// TwinCAT 3 PLC project DataProcessing
// ProgramVersion: 3.1.4023.0
// libraries:
//   Tc2_Standard, * (Beckhoff Automation GmbH)
//   Tc2_System, * (Beckhoff Automation GmbH)
//   Tc2_Utilities, * (Beckhoff Automation GmbH)
//   Tc3_EventLogger, * (Beckhoff Automation GmbH)
//   Tc3_Module, * (Beckhoff Automation GmbH)
// project tree:
//   DUTs/ FB_GetFaultWordsFromProtxConverter.TcPOU, FB_PrepareOutputVectorsToProTxConverter.TcPOU, FB_PrepareInputVectorsFromProTxCovnerter.TcPOU, FB_GetStatusWordsFromProTxConverter.TcPOU
//   Enumerations/ E_DriveProfile.TcDUT
//   EventLogger/FunctionBlocks/Common/ P_EventLogger.TcPOU, P_Timer.TcPOU
//   EventLogger/FunctionBlocks/ FB_EventMessage.TcPOU, FB_EventAlarm.TcPOU
//   GVLs/ ConfigurationParameters.TcGVL, RxAndTxData.TcGVL, StatusAndCommandWordsStructures.TcGVL, UtilityVariables.TcGVL
//   GVLs/ST_OutputVectorsToProTx/ ST_OutputVectorReal.TcDUT, ST_LcCommandWord_ProfiDrive.TcDUT, ST_McCommandWord_1_ProfiDrive.TcDUT, ST_McCommandWord_2_ProfiDrive.TcDUT
//   GVLs/ST_InputVectorsFromProTx/ST_FaultWords/ ST_LcFaultWord1.TcDUT, ST_LcFaultWord2.TcDUT, ST_LcFaultWord3.TcDUT, ST_LcFaultWord4.TcDUT, ST_McFaultWord1.TcDUT, ST_McFaultWord2.TcDUT, ST_McFaultWord3.TcDUT, ST_McFaultWord4.TcDUT
//   GVLs/ST_InputVectorsFromProTx/ ST_LcStatusWord_2_ProfiDrive.TcDUT, ST_McStatusWord_2_ProfiDrive.TcDUT, ST_LcStatusWord_1_ProfiDrive.TcDUT, ST_McStatusWord_1_ProfiDrive.TcDUT, ST_OutputVectorReal1.TcDUT
//   / PlcTask.TcTTO
//   POUs/ MAIN.TcPOU
// real-time tasks:
//   TASK PlcTask: cycle T#1ms, priority 20, ADS port 350

CONFIGURATION DataProcessing
    RESOURCE PLC ON TwinCAT3
        TASK PlcTask(INTERVAL := T#1ms, PRIORITY := 20);
        PROGRAM MAIN WITH PlcTask : MAIN;
    END_RESOURCE
END_CONFIGURATION

// ---- Enumerations/E_DriveProfile.TcDUT
{attribute 'qualified_only'}
{attribute 'strict'}
TYPE E_DriveProfile :
(
	CiA402 		:= 1,
	CAN 		:= 2,
	ProfiDrive  := 3
	
) := ProfiDrive;
END_TYPE

// ---- GVLs/ST_OutputVectorsToProTx/ST_OutputVectorReal.TcDUT
TYPE ST_OutputVectorReal :
STRUCT
	OutputPDO_1 			: REAL; // LC Iq_ref and  MC torque or current
	OutputPDO_2 			: REAL; // MC speed or voltge
	OutputPDO_3				: REAL; // Mc act. torque or power
	OutputPDO_4				: REAL; // MC Ext Torque Limmit_motor or Charge current limmit
	OutputPDO_5				: REAL; // MC Ext Torque Limmit_gen or Discharge current limmit
	OutputPDO_6				: REAL; // MC Speed regulation bias and Cable resistor in Ohm
	OutputPDO_7				: REAL; // MC Speed limmit and Max output votltage switch off value in V
	OutputPDO_8				: REAL; // MC Jrequest and and Min output votltage switch off value in V
	OutputPDO_9				: REAL; // MC Max output current switch off value in A and ETPS value for number of cylinders
	OutputPDO_10			: REAL;	// MC Min output current switch off value in A and scaled ETPS torque M1
END_STRUCT
END_TYPE

// ---- GVLs/ST_OutputVectorsToProTx/ST_LcCommandWord_ProfiDrive.TcDUT
TYPE ST_LcCommandWord_ProfiDrive :
STRUCT
	Bit00_OnOff 						: BOOL;
	Bit01_DriveRelease					: BOOL;
	Bit02_uu 							: BOOL;
	Bit03_PulseRelease 					: BOOL;
	Bit04_uu							: BOOL;
	Bit05_uu							: BOOL;
	Bit06_uu							: BOOL;
	Bit07_Quit							: BOOL;
	Bit08_uu							: BOOL;
	Bit09_uu							: BOOL;
	Bit10_ControlByPLC					: BOOL;
	Bit11_ParSetChangeOverBit00			: BOOL;
	Bit12_ParSetChangeOverBit01			: BOOL;
	Bit13_ParSetChangeOverBit02			: BOOL;
	Bit14_ParSetChangeOverBit03			: BOOL;
	Bit15_MainAliveToggle				: BOOL;

END_STRUCT
END_TYPE

// ---- GVLs/ST_OutputVectorsToProTx/ST_McCommandWord_1_ProfiDrive.TcDUT
TYPE ST_McCommandWord_1_ProfiDrive :
STRUCT
	Bit00_OnOff 					: BOOL;
	Bit01_DriveRelease				: BOOL;
	Bit02_FastStop 					: BOOL; // FALCE - forces QuickStop
	Bit03_PulceRelease 				: BOOL;
	Bit04_EnableRump				: BOOL; // TRUE - Select ramp output as reference; FALCE - select other reference source - may be zero 
	Bit05_UnlockRump				: BOOL; // TRUE - Ramp output shall follow ramp input; FALCE - Ramp output shall be locked to current output value
	Bit06_Forward					: BOOL;
	Bit07_Quit						: BOOL;
	Bit08_Inching1					: BOOL;
	Bit09_Inching2					: BOOL;
	Bit10_ControlByPlc				: BOOL;
	Bit11_ParSetChangeOverBit00		: BOOL;
	Bit12_ParSetChangeOverBit01		: BOOL;
	Bit13_ParSetChangeOverBit02		: BOOL;
	Bit14_ParSetChangeOverBit03		: BOOL;
	Bit15_MainAliveToggle			: BOOL;	
END_STRUCT
END_TYPE

// ---- GVLs/ST_OutputVectorsToProTx/ST_McCommandWord_2_ProfiDrive.TcDUT
TYPE ST_McCommandWord_2_ProfiDrive :
STRUCT
	Bit00_IntegratorSpeedCtrlDisable	: BOOL;
	Bit01_TorqueControlModeActive		: BOOL;
	Bit02_GainSpeedcontrolChangeover 	: BOOL;
	Bit03_Drooping 						: BOOL;
	Bit04_TorqueControlEnable			: BOOL;
	Bit05_TorqueReferenceEnable			: BOOL;
	Bit06_EtpsEnable					: BOOL;
	Bit07_EtpsInputSourceSelect			: BOOL;
	Bit08_InertiaCompensationenable		: BOOL;
	Bit09_ExternalMotorFanOff			: BOOL;
	Bit10_uu							: BOOL;
	Bit11_uu							: BOOL;
	Bit12_Reverce						: BOOL;
	Bit13_BrakeControl					: BOOL;
	Bit14_BrakeTestMode					: BOOL;
	Bit15_InternalAliveToggle			: BOOL;	
END_STRUCT
END_TYPE

// ---- GVLs/ST_InputVectorsFromProTx/ST_FaultWords/ST_LcFaultWord1.TcDUT
TYPE ST_LcFaultWord1 :
STRUCT
	Bit00_FaultInputAryEcat 	: BOOL;
	Bit01_FPGA					: BOOL;
	Bit02_Watchdog 				: BOOL;
	Bit03_UdcMax 				: BOOL;
	Bit04_uu					: BOOL;
	Bit05_uu					: BOOL;
	Bit06_uu					: BOOL;
	Bit07_uu					: BOOL;
	Bit08_UceFault				: BOOL;
	Bit09_uu					: BOOL;
	Bit10_uu					: BOOL;
	Bit11_uu					: BOOL;
	Bit12_uu					: BOOL;
	Bit13_uu					: BOOL;
	Bit14_uu					: BOOL;
	Bit15_uu					: BOOL;	
END_STRUCT
END_TYPE

// ---- GVLs/ST_InputVectorsFromProTx/ST_FaultWords/ST_LcFaultWord2.TcDUT
TYPE ST_LcFaultWord2 :
STRUCT
	Bit00_PibSupply 				: BOOL;
	Bit01_MeasurementConnectorLoop	: BOOL;
	Bit02_FaultLoop 				: BOOL;
	Bit03_AmplifierConnector 		: BOOL;
	Bit04_TermSupply 				: BOOL;
	Bit05_Overcurrent 				: BOOL;
	Bit06_ShortCircuit 				: BOOL;
	Bit07_DcConnection				: BOOL;
	Bit08_ThHSMax					: BOOL;
	Bit09_ShortCircuit24V			: BOOL;
	Bit10_FieldBus					: BOOL;
	Bit11_FLinkRxMc					: BOOL;
	Bit12_EarthFault				: BOOL;
	Bit13_UdcMin					: BOOL;
	Bit14_uu						: BOOL;
	Bit15_ExtFault					: BOOL;	
END_STRUCT
END_TYPE

// ---- GVLs/ST_InputVectorsFromProTx/ST_FaultWords/ST_LcFaultWord3.TcDUT
TYPE ST_LcFaultWord3 :
STRUCT
	Bit00_ULineVoltage 				: BOOL;
	Bit01_ULineMeasurement			: BOOL;
	Bit02_AcFuse	 				: BOOL;
	Bit03_FbLineContactor	 		: BOOL;
	Bit04_Charging	 				: BOOL;
	Bit05_LineFilter 				: BOOL;
	Bit06_uu		 				: BOOL;
	Bit07_uu						: BOOL;
	Bit08_uu						: BOOL;
	Bit09_uu						: BOOL;
	Bit10_uu						: BOOL;
	Bit11_uu						: BOOL;
	Bit12_uu						: BOOL;
	Bit13_uu						: BOOL;
	Bit14_uu						: BOOL;
	Bit15_uu						: BOOL;	
END_STRUCT
END_TYPE

// ---- GVLs/ST_InputVectorsFromProTx/ST_FaultWords/ST_LcFaultWord4.TcDUT
TYPE ST_LcFaultWord4 :
STRUCT
	Bit00_NTC 						: BOOL;
	Bit01_ThHsMin					: BOOL;
	Bit02_CoolingSystem 			: BOOL;
	Bit03_ControllerCabinetFan 		: BOOL;
	Bit04_ConverterCubiceOvertemp 	: BOOL;
	Bit05_CubicleAuxSupply 			: BOOL;
	Bit06_uu 						: BOOL;
	Bit07_uu						: BOOL;
	Bit08_uu						: BOOL;
	Bit09_FeedInCubicleOvertemp		: BOOL;
	Bit10_TrafoOvertemp				: BOOL;
	Bit11_Isolation					: BOOL;
	Bit12_uu						: BOOL;
	Bit13_uu						: BOOL;
	Bit14_uu						: BOOL;
	Bit15_uu						: BOOL;	
END_STRUCT
END_TYPE

// ---- GVLs/ST_InputVectorsFromProTx/ST_FaultWords/ST_McFaultWord1.TcDUT
TYPE ST_McFaultWord1 :
STRUCT
	Bit00_FaultInputAryEcat 	: BOOL;
	Bit01_FPGA					: BOOL;
	Bit02_Watchdog 				: BOOL;
	Bit03_UdcMax 				: BOOL;
	Bit04_uu					: BOOL;
	Bit05_uu					: BOOL;
	Bit06_uu					: BOOL;
	Bit07_uu					: BOOL;
	Bit08_UceFault				: BOOL;
	Bit09_uu					: BOOL;
	Bit10_uu					: BOOL;
	Bit11_uu					: BOOL;
	Bit12_uu					: BOOL;
	Bit13_uu					: BOOL;
	Bit14_uu					: BOOL;
	Bit15_uu					: BOOL;	
END_STRUCT
END_TYPE

// ---- GVLs/ST_InputVectorsFromProTx/ST_FaultWords/ST_McFaultWord2.TcDUT
TYPE ST_McFaultWord2 :
STRUCT
	Bit00_PibSupply 				: BOOL;
	Bit01_MeasurementConnectorLoop	: BOOL;
	Bit02_FaultLoop 				: BOOL;
	Bit03_AmplifierConnector 		: BOOL;
	Bit04_TermSupply 				: BOOL;
	Bit05_Overcurrent 				: BOOL;
	Bit06_ShortCircuit 				: BOOL;
	Bit07_DcConnection				: BOOL;
	Bit08_ThHSMax					: BOOL;
	Bit09_ShortCircuit24V			: BOOL;
	Bit10_FieldBus					: BOOL;
	Bit11_FLinkRxMc					: BOOL;
	Bit12_EarthFault				: BOOL;
	Bit13_UdcMin					: BOOL;
	Bit14_uu						: BOOL;
	Bit15_ExtFault					: BOOL;	
END_STRUCT
END_TYPE

// ---- GVLs/ST_InputVectorsFromProTx/ST_FaultWords/ST_McFaultWord3.TcDUT
TYPE ST_McFaultWord3 :
STRUCT
	Bit00_EncoderFault 				: BOOL;
	Bit01_BlockFault				: BOOL;
	Bit02_OverspeedFault			: BOOL;
	Bit03_BrakeFault		 		: BOOL;
	Bit04_InterlockRotating			: BOOL;
	Bit05_DcOutputSwitches			: BOOL;
	Bit06_DcOutputOfRange			: BOOL;
	Bit07_DcSwitchOnSequence		: BOOL;
	Bit08_uu						: BOOL;
	Bit09_uu						: BOOL;
	Bit10_uu						: BOOL;
	Bit11_uu						: BOOL;
	Bit12_uu						: BOOL;
	Bit13_uu						: BOOL;
	Bit14_uu						: BOOL;
	Bit15_uu						: BOOL;	
END_STRUCT
END_TYPE

// ---- GVLs/ST_InputVectorsFromProTx/ST_FaultWords/ST_McFaultWord4.TcDUT
TYPE ST_McFaultWord4 :
STRUCT
	Bit00_NTC 						: BOOL;
	Bit01_ThHsMin					: BOOL;
	Bit02_uu			 			: BOOL;
	Bit03_ControllerCabinetFan 		: BOOL;
	Bit04_ConverterCubiceOvertemp 	: BOOL;
	Bit05_CubicleAuxSupply 			: BOOL;
	Bit06_MotorTemp					: BOOL;
	Bit07_uu						: BOOL;
	Bit08_FrequLock					: BOOL;
	Bit09_ConverterOverload			: BOOL;
	Bit10_uu						: BOOL;
	Bit11_uu						: BOOL;
	Bit12_uu						: BOOL;
	Bit13_uu						: BOOL;
	Bit14_uu						: BOOL;
	Bit15_uu						: BOOL;	
END_STRUCT
END_TYPE

// ---- GVLs/ST_InputVectorsFromProTx/ST_LcStatusWord_2_ProfiDrive.TcDUT
TYPE ST_LcStatusWord_2_ProfiDrive :
STRUCT
	Bit00_FaultB					: BOOL;
	Bit01_FaultC 					: BOOL;
	Bit02_FaultC 					: BOOL;
	Bit03_FaultDWarning 			: BOOL;
	Bit04_TrafoOvertempWarning		: BOOL;
	Bit05_TrafoInsolationWarning	: BOOL;
	Bit06_uu						: BOOL;
	Bit07_uu						: BOOL;
	Bit08_uu						: BOOL;
	Bit09_uu						: BOOL;
	Bit10_ThHSWarning				: BOOL;
	Bit11_ThHSMaxWarning			: BOOL;
	Bit12_ParSetBit00				: BOOL;
	Bit13_ParSetBit01				: BOOL;
	Bit14_ParSetBit02				: BOOL;
	Bit15_ParSetBit03				: BOOL;	
END_STRUCT
END_TYPE

// ---- GVLs/ST_InputVectorsFromProTx/ST_McStatusWord_2_ProfiDrive.TcDUT
TYPE ST_McStatusWord_2_ProfiDrive :
STRUCT
	Bit00_FaultB					: BOOL;
	Bit01_FaultC 					: BOOL;
	Bit02_FaultC 					: BOOL;
	Bit03_FaultDWarning 			: BOOL;
	Bit04_MRegActive				: BOOL;
	Bit05_torqueRegEnable			: BOOL;
	Bit06_ConverterI2tLinitWarning	: BOOL;
	Bit07_ConverterI2tLinitActive	: BOOL;
	Bit08_MotorI2tLinitWarning		: BOOL;
	Bit09_MotorI2tLinitActive		: BOOL;
	Bit10_ThHSWarning				: BOOL;
	Bit11_ThHSMaxWarning			: BOOL;
	Bit12_windingTempWarning		: BOOL;
	Bit13_BearingTempWarning		: BOOL;
	Bit14_Forward					: BOOL;
	Bit15_Reverse					: BOOL;	
END_STRUCT
END_TYPE

// ---- GVLs/ST_InputVectorsFromProTx/ST_LcStatusWord_1_ProfiDrive.TcDUT
TYPE ST_LcStatusWord_1_ProfiDrive :
STRUCT
	Bit00_StateReady			: BOOL;
	Bit01_StateOn 				: BOOL;
	Bit02_CtrlRun 				: BOOL;
	Bit03_CollFault 			: BOOL;
	Bit04_DriveReleaseActive	: BOOL;
	Bit05_StatePowerOk			: BOOL;
	Bit06_StateDisable			: BOOL;
	Bit07_Warning				: BOOL;
	Bit08_PhaseLoss				: BOOL;
	Bit09_BusSelected			: BOOL;
	Bit10_uu					: BOOL;
	Bit11_uu					: BOOL;
	Bit12_ReleaseMc				: BOOL;
	Bit13_StateTestModeOn		: BOOL;
	Bit14_InternalAliveToggle	: BOOL;
	Bit15_MainAliveToggle		: BOOL;	
END_STRUCT
END_TYPE

// ---- GVLs/ST_InputVectorsFromProTx/ST_McStatusWord_1_ProfiDrive.TcDUT
TYPE ST_McStatusWord_1_ProfiDrive :
STRUCT
	Bit00_StateReady			: BOOL;
	Bit01_StateOn 				: BOOL;
	Bit02_CtrlRun 				: BOOL;
	Bit03_CollFault 			: BOOL;
	Bit04_DriveReleaseActive	: BOOL;
	Bit05_StateFastStop			: BOOL;
	Bit06_StateDisable			: BOOL;
	Bit07_Warning				: BOOL;
	Bit08_SpeedCtrlLimited		: BOOL;
	Bit09_BusSelected			: BOOL;
	Bit10_XnIsEqualToWn			: BOOL;
	Bit11_WiqTLimited			: BOOL;
	Bit12_XnIsEqualToZero		: BOOL;
	Bit13_NCtrlenable			: BOOL;
	Bit14_ExtrnalTorqueRelease	: BOOL;
	Bit15_MainAliveToggle		: BOOL;	
END_STRUCT
END_TYPE

// ---- GVLs/ST_InputVectorsFromProTx/ST_OutputVectorReal1.TcDUT
TYPE ST_OutputVectorReal1 :
STRUCT
	Element00_LcActualVauleOfUdc 					: REAL;
	Element01_LcSmoothedConverterCurrent 			: REAL;
	Element02_LcMeasuredMainsVoltage				: REAL;
	Element03_LcActualHeatsinkTemp					: REAL;
	Element04_LcMinimumHeatsinkTemp					: REAL;
 	Element05_LcCurrentReferenceValueInDAxis		: REAL;
	Element06_LcReactiveCurrentFerenceValue			: REAL;
	Element07_LcFilteredLineFrequency				: REAL;
	Element08_LcActivePowerOfLineConverter			: REAL;
	Element09_LcReactivePowerOfLineConverter		: REAL;
	Element10_LcTestValue							: REAL;
	Element11_McSumOfPowerReference					: REAL;
	Element12_McSmoothedConverterCurrent			: REAL;
	Element13_McInverterOutputVoltage				: REAL;
	Element14_McSumOfTorqueReference				: REAL;
	Element15_McMeasuredOrEstimatedSpeed			: REAL;
	Element16_McActualHeatsinkTemp					: REAL;
	Element17_McMinimumHeatsinkTemp					: REAL;
	Element18_McMaxvalueOfTwoMeasuredBearingTemp	: REAL;
	Element19_McMaxvalueOfThreeMeasuredWindingTemp	: REAL;
	Element20_McReferenceValueOfIq					: REAL;	
	Element21_McActualValueOfIq						: REAL;	
	Element22_McReferenceValueOfId					: REAL;	
	Element23_McActualValueOfId						: REAL;
	Element24_McIntegratorOutputOfConverterI2t		: REAL;
	Element25_McIntegratorOutputOfMotorI2t			: REAL;
	Element26_McTestValue							: REAL;			
END_STRUCT
END_TYPE

// ---- GVLs/ConfigurationParameters.TcGVL
{attribute 'qualified_only'}
VAR_GLOBAL
	
	(* Configuration Parameters *)
	
	LcCmdDriveProfile : E_DriveProfile;
	
END_VAR

// ---- GVLs/RxAndTxData.TcGVL
{attribute 'qualified_only'}
VAR_GLOBAL

	(* Recieved Integer PDOs From ProTX, Status Words *)
	nLcStatusWord_1 		AT %I* : UDINT; // LC Status Word 1
	nLcStatusWord_2 		AT %I* : UDINT; // LC Status Word 2
	nMcStatusWord_1 		AT %I* : UDINT; // LC Status Word 1
	nMcStatusWord_2 		AT %I* : UDINT; // LC Status Word 2
	
	
	(* Recieved Integer PDOs From ProTX, Fault Words *)
	nLcFaultWord1 			AT %I* : UDINT; // Drive fault category B
	nLcFaultWord2 			AT %I* : UDINT; // Drive fault category C #1
	nLcFaultWord3 			AT %I* : UDINT; // Drive fault category C #2
	nLcFaultWord4 			AT %I* : UDINT; // Drive fault category D
	nMcFaultWord1 			AT %I* : UDINT; // Drive fault category B
	nMcFaultWord2 			AT %I* : UDINT; // Drive fault category C #1
	nMcFaultWord3 			AT %I* : UDINT; // Drive fault category C #2
	nMcFaultWord4 			AT %I* : UDINT; // Drive fault category D
	

	(* Recieved Real PDOs From ProTx *)
	
	TxRealPdo01 			AT %I* : REAL; 
	TxRealPdo02 			AT %I* : REAL;
	TxRealPdo03 			AT %I* : REAL;
	TxRealPdo04 			AT %I* : REAL;
	TxRealPdo05 			AT %I* : REAL;
	TxRealPdo06 			AT %I* : REAL;
	TxRealPdo07 			AT %I* : REAL;
	TxRealPdo08 			AT %I* : REAL;
	TxRealPdo09 			AT %I* : REAL;
	TxRealPdo10 			AT %I* : REAL;
	TxRealPdo11 			AT %I* : REAL;
	TxRealPdo12 			AT %I* : REAL;
	TxRealPdo13 			AT %I* : REAL;
	TxRealPdo14 			AT %I* : REAL;
	TxRealPdo15 			AT %I* : REAL;
	TxRealPdo16 			AT %I* : REAL;
	TxRealPdo17 			AT %I* : REAL;
	TxRealPdo18 			AT %I* : REAL;
	TxRealPdo19 			AT %I* : REAL;
	TxRealPdo20 			AT %I* : REAL;
	TxRealPdo21 			AT %I* : REAL;
	TxRealPdo22 			AT %I* : REAL;
	
	(*  Send Integer variable to ProTx, Command Words, lincked to IO *)
	
	nLcCommandWord 			AT %Q* : UDINT; 	// LC Command Word
	nMcCommandWord_1 		AT %Q* : UDINT; 	// MC Main Command Word
	nMcCommandWord_2		AT %Q* : UDINT; 	// MC Application Command Word

	(* Send Real variables to ProTX, lincked to IO *)
	
	RxRealPdo01 			AT %Q* : REAL; // LC Iq_ref and  MC torque or current
	RxRealPdo02 			AT %Q* : REAL; // MC speed or voltge
	RxRealPdo03 			AT %Q* : REAL; // Mc act. torque or power
	RxRealPdo04 			AT %Q* : REAL; // MC Ext Torque Limmit_motor or Charge current limmit
	RxRealPdo05				AT %Q* : REAL; // MC Ext Torque Limmit_gen or Discharge current limmit
	RxRealPdo06 			AT %Q* : REAL; // MC Speed regulation bias and Cable resistor in Ohm
	RxRealPdo07 			AT %Q* : REAL; // MC Speed limmit and Max output votltage switch off value in V
	RxRealPdo08 			AT %Q* : REAL; // MC Jrequest and and Min output votltage switch off value in V
	RxRealPdo09 			AT %Q* : REAL; // MC Max output current switch off value in A and ETPS value for number of cylinders
	RxRealPdo10 			AT %Q* : REAL; // MC Min output current switch off value in A and scaled ETPS torque M1
	
END_VAR

// ---- GVLs/StatusAndCommandWordsStructures.TcGVL
{attribute 'qualified_only'}
VAR_GLOBAL
	(* Recieved Status and Fault Words*)
	stLcStatusWord_1 	: ST_LcStatusWord_1_ProfiDrive;
	stLcStatusWord_2 	: ST_LcStatusWord_2_ProfiDrive;
	stMcStatusWord_1 	: ST_McStatusWord_1_ProfiDrive;
	stMcStatusWord_2 	: ST_McStatusWord_2_ProfiDrive;
	
	stLcFaultWord1 		: ST_LcFaultWord1;
	stLcFaultWord2 		: ST_LcFaultWord2;
	stLcFaultWord3 		: ST_LcFaultWord3;
	stLcFaultWord4 		: ST_LcFaultWord4;
	stMcFaultWord1 		: ST_McFaultWord1;
	stMcFaultWord2 		: ST_McFaultWord2;
	stMcFaultWord3 		: ST_McFaultWord3;
	stMcFaultWord4 		: ST_McFaultWord4;
END_VAR

// ---- GVLs/UtilityVariables.TcGVL
{attribute 'qualified_only'}
VAR_GLOBAL
	nEventsInEventLogger : INT; // Number of events on event logger buffer
END_VAR

// ---- POUs/MAIN.TcPOU
PROGRAM MAIN
VAR
    
    fbPrepareOutputVectorsToProTxConverter      : FB_PrepareOutputVectorsToProTxConverter;
//    fbPrepareInputVectorsFromProTxCovnerter     : FB_PrepareInputVectorsFromProTxCovnerter;
//    fbGetFaultWordsFromProtxConverter           : FB_GetFaultWordsFromProtxConverter;
//    fbGetStatusWordsFromProTxConverter          : FB_GetStatusWordsFromProTxConverter;    
    
    stOutputVectorReal                          : ST_OutputVectorReal;
    stLcCommandWord_ProfiDrive                  : ST_LcCommandWord_ProfiDrive;
    stMcCommandWord_1_ProfiDrive                : ST_McCommandWord_1_ProfiDrive;
    stMcCommandWord_2_ProfiDrive                : ST_McCommandWord_2_ProfiDrive;
    
    nLcDriveProfile                             : E_DriveProfile; // Default is ProfiDrive
    nMcDriveProfile                             : E_DriveProfile; // Default is ProfiDrive
    
    bOnOff                                      : BOOL;
    bDriveRelease                               : BOOL;
    bFastStop                                   : BOOL := TRUE;
    bPulseRelease                               : BOOL;
    bForward                                    : BOOL;
    bReverse                                    : BOOL;
    bControlByPlc                               : BOOL;
     
END_VAR

P_EventLogger();
P_Timer();

stMcCommandWord_1_ProfiDrive.Bit15_MainAliveToggle  := P_Timer.bPulse05s;
stMcCommandWord_1_ProfiDrive.Bit02_FastStop         := bFastStop;
stMcCommandWord_1_ProfiDrive.Bit01_DriveRelease     := bDriveRelease;
stMcCommandWord_1_ProfiDrive.Bit00_OnOff            := bOnOff;
stMcCommandWord_1_ProfiDrive.Bit03_PulceRelease     := bPulseRelease;
stMcCommandWord_1_ProfiDrive.Bit06_Forward          := bForward;
stMcCommandWord_2_ProfiDrive.Bit12_Reverce          := bReverse;
stMcCommandWord_1_ProfiDrive.Bit10_ControlByPlc     := bControlByPlc;

 

fbPrepareOutputVectorsToProTxConverter(
    stOutputVectorReal  := stOutputVectorReal, 
    stLcCommandWord     := stLcCommandWord_ProfiDrive, 
    stMcCommandWord_1   := stMcCommandWord_1_ProfiDrive, 
    stMcCommandWord_2   := stMcCommandWord_2_ProfiDrive, 
    nLcDriveProfile     := nLcDriveProfile, 
    nMcDriveProfile     := nMcDriveProfile);

END_PROGRAM

// ---- DUTs/FB_PrepareOutputVectorsToProTxConverter.TcPOU
FUNCTION_BLOCK FB_PrepareOutputVectorsToProTxConverter
VAR_INPUT
	stOutputVectorReal 				: ST_OutputVectorReal;
	stLcCommandWord 				: ST_LcCommandWord_ProfiDrive;
	stMcCommandWord_1 				: ST_McCommandWord_1_ProfiDrive;
	stMcCommandWord_2		 		: ST_McCommandWord_2_ProfiDrive;
	nLcDriveProfile 				: E_DriveProfile;
	nMcDriveProfile 				: E_DriveProfile;
END_VAR 
VAR
	wLcCommandWord 					: WORD;
	wMcCommandWord_1 				: WORD;
	wMcCommandWord_2		 		: WORD;
END_VAR


/// Converting LC Command Word From Structure to UDINT {{{
IF 	nLcDriveProfile = 3 THEN
	wLcCommandWord.0 := stLcCommandWord.Bit00_OnOff;
	wLcCommandWord.1 := stLcCommandWord.Bit01_DriveRelease;
	wLcCommandWord.2 := stLcCommandWord.Bit02_uu;
	wLcCommandWord.3 := stLcCommandWord.Bit03_PulseRelease;
	wLcCommandWord.4 := stLcCommandWord.Bit04_uu;
	wLcCommandWord.5 := stLcCommandWord.Bit05_uu;
	wLcCommandWord.6 := stLcCommandWord.Bit06_uu;
	wLcCommandWord.7 := stLcCommandWord.Bit07_Quit;
	wLcCommandWord.8 := stLcCommandWord.Bit08_uu;
	wLcCommandWord.9 := stLcCommandWord.Bit09_uu;
	wLcCommandWord.10 := stLcCommandWord.Bit10_ControlByPLC;
	wLcCommandWord.11 := stLcCommandWord.Bit11_ParSetChangeOverBit00;
	wLcCommandWord.12 := stLcCommandWord.Bit12_ParSetChangeOverBit01;
	wLcCommandWord.13 := stLcCommandWord.Bit13_ParSetChangeOverBit02;
	wLcCommandWord.14 := stLcCommandWord.Bit14_ParSetChangeOverBit03;
	wLcCommandWord.15 := stLcCommandWord.Bit15_MainAliveToggle;
END_IF
	
	RxAndTxData.nLcCommandWord := TO_UDINT(wLcCommandWord);
///}}}

/// Converting MC Command Word_1 From Structure to UDINT {{{
IF 	nMcDriveProfile = 3 THEN
	wMcCommandWord_1.0 := stMcCommandWord_1.Bit00_OnOff;
	wMcCommandWord_1.1 := stMcCommandWord_1.Bit01_DriveRelease;
	wMcCommandWord_1.2 := stMcCommandWord_1.Bit02_FastStop;
	wMcCommandWord_1.3 := stMcCommandWord_1.Bit03_PulceRelease;
	wMcCommandWord_1.4 := stMcCommandWord_1.Bit04_EnableRump;
	wMcCommandWord_1.5 := stMcCommandWord_1.Bit05_UnlockRump;
	wMcCommandWord_1.6 := stMcCommandWord_1.Bit06_Forward;
	wMcCommandWord_1.7 := stMcCommandWord_1.Bit07_Quit;
	wMcCommandWord_1.8 := stMcCommandWord_1.Bit08_Inching1;
	wMcCommandWord_1.9 := stMcCommandWord_1.Bit09_Inching2;
	wMcCommandWord_1.10 := stMcCommandWord_1.Bit10_ControlByPlc;
	wMcCommandWord_1.11 := stMcCommandWord_1.Bit11_ParSetChangeOverBit00;
	wMcCommandWord_1.12 := stMcCommandWord_1.Bit12_ParSetChangeOverBit01;
	wMcCommandWord_1.13 := stMcCommandWord_1.Bit13_ParSetChangeOverBit02;
	wMcCommandWord_1.14 := stMcCommandWord_1.Bit14_ParSetChangeOverBit03;
	wMcCommandWord_1.15 := stMcCommandWord_1.Bit15_MainAliveToggle;
END_IF
	
	RxAndTxData.nMcCommandWord_1 := TO_UDINT(wMcCommandWord_1);
///}}}

/// Converting MC Command Word_2 From Structure to UDINT {{{
IF 	nMcDriveProfile = 3 THEN
	wMcCommandWord_2.0 := stMcCommandWord_2.Bit00_IntegratorSpeedCtrlDisable;
	wMcCommandWord_2.1 := stMcCommandWord_2.Bit01_TorqueControlModeActive;
	wMcCommandWord_2.2 := stMcCommandWord_2.Bit02_GainSpeedcontrolChangeover;
	wMcCommandWord_2.3 := stMcCommandWord_2.Bit03_Drooping;
	wMcCommandWord_2.4 := stMcCommandWord_2.Bit04_TorqueControlEnable;
	wMcCommandWord_2.5 := stMcCommandWord_2.Bit05_TorqueReferenceEnable;
	wMcCommandWord_2.6 := stMcCommandWord_2.Bit06_EtpsEnable;
	wMcCommandWord_2.7 := stMcCommandWord_2.Bit07_EtpsInputSourceSelect;
	wMcCommandWord_2.8 := stMcCommandWord_2.Bit08_InertiaCompensationenable;
	wMcCommandWord_2.9 := stMcCommandWord_2.Bit09_ExternalMotorFanOff;
	wMcCommandWord_2.10 := stMcCommandWord_2.Bit10_uu;
	wMcCommandWord_2.11 := stMcCommandWord_2.Bit11_uu;
	wMcCommandWord_2.12 := stMcCommandWord_2.Bit12_Reverce;
	wMcCommandWord_2.13 := stMcCommandWord_2.Bit13_BrakeControl;
	wMcCommandWord_2.14 := stMcCommandWord_2.Bit14_BrakeTestMode;
	wMcCommandWord_2.15 := stMcCommandWord_2.Bit15_InternalAliveToggle;
END_IF

	RxAndTxData.nMcCommandWord_2 := TO_UDINT(wMcCommandWord_2);
///}}}

/// Converting Output Real PDOs to IO Linked  Variable {{{	
	RxAndTxData.RxRealPdo01 := stOutputVectorReal.OutputPDO_1;
	RxAndTxData.RxRealPdo02 := stOutputVectorReal.OutputPDO_2;
	RxAndTxData.RxRealPdo03 := stOutputVectorReal.OutputPDO_3;
	RxAndTxData.RxRealPdo04 := stOutputVectorReal.OutputPDO_4;
	RxAndTxData.RxRealPdo05 := stOutputVectorReal.OutputPDO_5;
	RxAndTxData.RxRealPdo06 := stOutputVectorReal.OutputPDO_6;
	RxAndTxData.RxRealPdo07 := stOutputVectorReal.OutputPDO_7;
	RxAndTxData.RxRealPdo08 := stOutputVectorReal.OutputPDO_8;
	RxAndTxData.RxRealPdo09 := stOutputVectorReal.OutputPDO_9;
	RxAndTxData.RxRealPdo10 := stOutputVectorReal.OutputPDO_10;
///}}}

END_FUNCTION_BLOCK

// ---- EventLogger/FunctionBlocks/Common/P_EventLogger.TcPOU
PROGRAM P_EventLogger
VAR
	fbEventlogger 								: FB_TcEventLogger;
	bClearAlarms 								: BOOL;
	bConfirmAlarms 								: BOOL;
	bClearLoggedEvents							: BOOL;
	bClearLoggedEventsAtInitialization			: BOOL := TRUE;
	bExportLoggedEvents							: BOOL;
	fbRtExport									: R_TRIG;
	fbLcSignalFaling							: ARRAY[0..30] OF F_TRIG;
	fbMcSignalFalingCommand						: ARRAY[0..30] OF F_TRIG;
	fbMcSignalFalingStatus						: ARRAY[0..35] OF F_TRIG;
	fbCsvExportSetting 							: FB_TcEventCsvExportSettings;
	fbExportFilter								: FB_TcEventfilter;
	sExportFileName								: STRING := 'c:\temp\Eventlogger-export.csv';
	
	fbLcControlCommandEvents 					: ARRAY[0..50] OF FB_EventMessage;
	fbMcControlCommandEvents					: ARRAY[0..50] OF FB_EventMessage;
	fbMcStatusEvents							: ARRAY[0..65] OF FB_EventMessage;
	
	
	hr											: HRESULT;
	hrLastError									: HRESULT;

	bError 	: BOOL;
	hrErrorCode 	: HRESULT;
	nFuulCounter : INT := 0; 
	nAskToCleanCounter : INT := 0;	
END_VAR

	
	// Instances of Action
	(* a_LcCommandEvents(); *)
	a_McCommandEvents();
	a_McStatusEvents();
	a_ExportLoggedEvents();
	a_ClearLoggedEvents();
	
	// Clear Event Logger Buffer At Initialisation
	IF bClearLoggedEventsAtInitialization THEN
		bClearLoggedEventsAtInitialization := FALSE;
		fbEventlogger.ClearLoggedEvents(0);
	END_IF
	
	// If Event Logger Buffer is Full then Export them in CSV File and Clear Event Logger Buffer
	IF UtilityVariables.nEventsInEventLogger >= 1000 THEN 
		bExportLoggedEvents := TRUE;
		bClearLoggedEvents := TRUE;
		UtilityVariables.nEventsInEventLogger := 0;
	END_IF

ACTION a_ClearEventCecheWhenFull:
// Stors an event CSV file and clears a PLC ceche when Eevent number is equal to 1000;
	IF UtilityVariables.nEventsInEventLogger = 10 THEN 
		bExportLoggedEvents := TRUE;
		fbEventlogger.ClearLoggedEvents(0);
		UtilityVariables.nEventsInEventLogger := 0;
	END_IF
END_ACTION

ACTION a_ClearLoggedEvents:
// Clear all logged events in PLC ceche
	IF bClearLoggedEvents THEN
		bClearLoggedEvents := FALSE;
		fbEventlogger.ClearLoggedEvents(0);
		fbEventlogger.ClearLoggedEvents(0);
	END_IF
END_ACTION

ACTION a_ExportLoggedEvents:
(* create file name *) 
	sExportFileName := CONCAT(CONCAT('C:\Temp\',P_Timer.sDateTime), '.csv');
	
(* CSV export logged events. Without filter all logged events will be exported *)
(* CSV file will be overwritten, an opened file fires an error *)

	fbRtExport(CLK := bExportLoggedEvents);
	IF bExportLoggedEvents THEN
		IF fbRtExport.Q THEN
			fbCsvExportSetting.Clear();
			fbCsvExportSetting.AddLanguage(1033, 'English');
		END_IF
		IF fbEventLogger.ExportLoggedEvents(sExportFileName, fbCsvExportSetting, hrErrorCode => hr) THEN 
			bExportLoggedEvents := FALSE;
		END_IF
	END_IF
END_ACTION

ACTION a_McCommandEvents:

(* Events coming from the MC commands *)

	fbMcControlCommandEvents[0](
		bEvent := RxAndTxData.nMcCommandWord_1.0,
		nEventID := 16#1000,
		sSource := 'Machince Converter Commands',
		sArgument1 := 'MC',
		sArgument2 := '1'
	);	
 	
	fbMcSignalFalingCommand[0](CLK := RxAndTxData.nMcCommandWord_1.0);
	fbMcControlCommandEvents[1](
		bEvent := fbMcSignalFalingCommand[0].Q,
		nEventID := 16#1001,
		sSource := 'Machince Converter Commands',
		sArgument1 := 'MC',
		sArgument2 := '1'
	);
	
	fbMcControlCommandEvents[2](
		bEvent := RxAndTxData.nMcCommandWord_1.1,
		nEventID := 16#1002,
		sSource := 'Machince Converter Commands',
		sArgument1 := 'MC',
		sArgument2 := '1'
	);	
 	
	fbMcSignalFalingCommand[1](CLK := RxAndTxData.nMcCommandWord_1.1);
	fbMcControlCommandEvents[3](
		bEvent := fbMcSignalFalingCommand[1].Q,
		nEventID := 16#1003,
		sSource := 'Machince Converter Commands',
		sArgument1 := 'MC',
		sArgument2 := '1'
	);
	
	fbMcControlCommandEvents[4](
		bEvent := RxAndTxData.nMcCommandWord_1.2,
		nEventID := 16#1004,
		sSource := 'Machince Converter Commands',
		sArgument1 := 'MC',
		sArgument2 := '1'
	);	
 	
	fbMcSignalFalingCommand[2](CLK := RxAndTxData.nMcCommandWord_1.2);
	fbMcControlCommandEvents[5](
		bEvent := fbMcSignalFalingCommand[2].Q,
		nEventID := 16#1005,
		sSource := 'Machince Converter Commands',
		sArgument1 := 'MC',
		sArgument2 := '1'
	);
	
	fbMcControlCommandEvents[6](
		bEvent := RxAndTxData.nMcCommandWord_1.3,
		nEventID := 16#1006,
		sSource := 'Machince Converter Commands',
		sArgument1 := 'MC',
		sArgument2 := '1'
	);	
 	
	fbMcSignalFalingCommand[3](CLK := RxAndTxData.nMcCommandWord_1.3);
	fbMcControlCommandEvents[7](
		bEvent := fbMcSignalFalingCommand[3].Q,
		nEventID := 16#1007,
		sSource := 'Machince Converter Commands',
		sArgument1 := 'MC',
		sArgument2 := '1'
	);
	
	fbMcControlCommandEvents[8](
		bEvent := RxAndTxData.nMcCommandWord_1.4,
		nEventID := 16#1008,
		sSource := 'Machince Converter Commands',
		sArgument1 := 'MC',
		sArgument2 := '1'
	);	
 	
	fbMcSignalFalingCommand[4](CLK := RxAndTxData.nMcCommandWord_1.4);
	fbMcControlCommandEvents[9](
		bEvent := fbMcSignalFalingCommand[4].Q,
		nEventID := 16#1009,
		sSource := 'Machince Converter Commands',
		sArgument1 := 'MC',
		sArgument2 := '1'
	);
	
	fbMcControlCommandEvents[10](
		bEvent := RxAndTxData.nMcCommandWord_1.5,
		nEventID := 16#100A,
		sSource := 'Machince Converter Commands',
		sArgument1 := 'MC',
		sArgument2 := '1'
	);	
 	
	fbMcSignalFalingCommand[5](CLK := RxAndTxData.nMcCommandWord_1.5);
	fbMcControlCommandEvents[11](
		bEvent := fbMcSignalFalingCommand[5].Q,
		nEventID := 16#100B,
		sSource := 'Machince Converter Commands',
		sArgument1 := 'MC',
		sArgument2 := '1'
	);
	
	fbMcControlCommandEvents[12](
		bEvent := RxAndTxData.nMcCommandWord_1.6,
		nEventID := 16#100C,
		sSource := 'Machince Converter Commands',
		sArgument1 := 'MC',
		sArgument2 := '1'
	);	
 	
	fbMcSignalFalingCommand[6](CLK := RxAndTxData.nMcCommandWord_1.6);
	fbMcControlCommandEvents[13](
		bEvent := fbMcSignalFalingCommand[6].Q,
		nEventID := 16#100D,
		sSource := 'Machince Converter Commands',
		sArgument1 := 'MC',
		sArgument2 := '1'
	);
	
	fbMcControlCommandEvents[14](
		bEvent := RxAndTxData.nMcCommandWord_1.7,
		nEventID := 16#100E,
		sSource := 'Machince Converter Commands',
		sArgument1 := 'MC',
		sArgument2 := '1'
	);	
 	
	fbMcSignalFalingCommand[7](CLK := RxAndTxData.nMcCommandWord_1.7);
	fbMcControlCommandEvents[15](
		bEvent := fbMcSignalFalingCommand[7].Q,
		nEventID := 16#100F,
		sSource := 'Machince Converter Commands',
		sArgument1 := 'MC',
		sArgument2 := '1'
	);
	
	fbMcControlCommandEvents[16](
		bEvent := RxAndTxData.nMcCommandWord_1.8,
		nEventID := 16#1010,
		sSource := 'Machince Converter Commands',
		sArgument1 := 'MC',
		sArgument2 := '1'
	);	
 	
	fbMcSignalFalingCommand[8](CLK := RxAndTxData.nMcCommandWord_1.8);
	fbMcControlCommandEvents[17](
		bEvent := fbMcSignalFalingCommand[8].Q,
		nEventID := 16#1011,
		sSource := 'Machince Converter Commands',
		sArgument1 := 'MC',
		sArgument2 := '1'
	);
	
	fbMcControlCommandEvents[18](
		bEvent := RxAndTxData.nMcCommandWord_1.9,
		nEventID := 16#1012,
		sSource := 'Machince Converter Commands',
		sArgument1 := 'MC',
		sArgument2 := '1'
	);	
 	
	fbMcSignalFalingCommand[9](CLK := RxAndTxData.nMcCommandWord_1.9);
	fbMcControlCommandEvents[19](
		bEvent := fbMcSignalFalingCommand[9].Q,
		nEventID := 16#1013,
		sSource := 'Machince Converter Commands',
		sArgument1 := 'MC',
		sArgument2 := '1'
	);
	
	fbMcControlCommandEvents[20](
		bEvent := RxAndTxData.nMcCommandWord_1.10,
		nEventID := 16#1014,
		sSource := 'Machince Converter Commands',
		sArgument1 := 'MC',
		sArgument2 := '1'
	);	
 	
	fbMcSignalFalingCommand[10](CLK := RxAndTxData.nMcCommandWord_1.10);
	fbMcControlCommandEvents[21](
		bEvent := fbMcSignalFalingCommand[10].Q,
		nEventID := 16#1015,
		sSource := 'Machince Converter Commands',
		sArgument1 := 'MC',
		sArgument2 := '1'
	);
	
	fbMcControlCommandEvents[22](
		bEvent := RxAndTxData.nMcCommandWord_2.0,
		nEventID := 16#1016,
		sSource := 'Machince Converter Commands',
		sArgument1 := 'MC',
		sArgument2 := '1'
	);	
 	
	fbMcSignalFalingCommand[11](CLK := RxAndTxData.nMcCommandWord_2.0);
	fbMcControlCommandEvents[23](
		bEvent := fbMcSignalFalingCommand[11].Q,
		nEventID := 16#1017,
		sSource := 'Machince Converter Commands',
		sArgument1 := 'MC',
		sArgument2 := '1'
	);

	fbMcControlCommandEvents[24](
		bEvent := RxAndTxData.nMcCommandWord_2.1,
		nEventID := 16#1018,
		sSource := 'Machince Converter Commands',
		sArgument1 := 'MC',
		sArgument2 := '1'
	);	
 	
	fbMcSignalFalingCommand[12](CLK := RxAndTxData.nMcCommandWord_2.1);
	fbMcControlCommandEvents[25](
		bEvent := fbMcSignalFalingCommand[12].Q,
		nEventID := 16#1019,
		sSource := 'Machince Converter Commands',
		sArgument1 := 'MC',
		sArgument2 := '1'
	);
	
	fbMcControlCommandEvents[26](
		bEvent := RxAndTxData.nMcCommandWord_2.2,
		nEventID := 16#101A,
		sSource := 'Machince Converter Commands',
		sArgument1 := 'MC',
		sArgument2 := '1'
	);	
 	
	fbMcSignalFalingCommand[13](CLK := RxAndTxData.nMcCommandWord_2.2);
	fbMcControlCommandEvents[27](
		bEvent := fbMcSignalFalingCommand[13].Q,
		nEventID := 16#101B,
		sSource := 'Machince Converter Commands',
		sArgument1 := 'MC',
		sArgument2 := '1'
	);
	
	fbMcControlCommandEvents[28](
		bEvent := RxAndTxData.nMcCommandWord_2.3,
		nEventID := 16#101C,
		sSource := 'Machince Converter Commands',
		sArgument1 := 'MC',
		sArgument2 := '1'
	);	
 	
	fbMcSignalFalingCommand[14](CLK := RxAndTxData.nMcCommandWord_2.3);
	fbMcControlCommandEvents[29](
		bEvent := fbMcSignalFalingCommand[14].Q,
		nEventID := 16#101D,
		sSource := 'Machince Converter Commands',
		sArgument1 := 'MC',
		sArgument2 := '1'
	);
	
	fbMcControlCommandEvents[30](
		bEvent := RxAndTxData.nMcCommandWord_2.4,
		nEventID := 16#101E,
		sSource := 'Machince Converter Commands',
		sArgument1 := 'MC',
		sArgument2 := '1'
	);	
 	
	fbMcSignalFalingCommand[15](CLK := RxAndTxData.nMcCommandWord_2.4);
	fbMcControlCommandEvents[31](
		bEvent := fbMcSignalFalingCommand[15].Q,
		nEventID := 16#101F,
		sSource := 'Machince Converter Commands',
		sArgument1 := 'MC',
		sArgument2 := '1'
	);
	
	fbMcControlCommandEvents[32](
		bEvent := RxAndTxData.nMcCommandWord_2.5,
		nEventID := 16#1020,
		sSource := 'Machince Converter Commands',
		sArgument1 := 'MC',
		sArgument2 := '1'
	);	
 	
	fbMcSignalFalingCommand[16](CLK := RxAndTxData.nMcCommandWord_2.5);
	fbMcControlCommandEvents[33](
		bEvent := fbMcSignalFalingCommand[16].Q,
		nEventID := 16#1021,
		sSource := 'Machince Converter Commands',
		sArgument1 := 'MC',
		sArgument2 := '1'
	);
	
	fbMcControlCommandEvents[34](
		bEvent := RxAndTxData.nMcCommandWord_2.6,
		nEventID := 16#1022,
		sSource := 'Machince Converter Commands',
		sArgument1 := 'MC',
		sArgument2 := '1'
	);	
 	
	fbMcSignalFalingCommand[17](CLK := RxAndTxData.nMcCommandWord_2.6);
	fbMcControlCommandEvents[35](
		bEvent := fbMcSignalFalingCommand[17].Q,
		nEventID := 16#1023,
		sSource := 'Machince Converter Commands',
		sArgument1 := 'MC',
		sArgument2 := '1'
	);
	
	fbMcControlCommandEvents[36](
		bEvent := RxAndTxData.nMcCommandWord_2.7,
		nEventID := 16#1024,
		sSource := 'Machince Converter Commands',
		sArgument1 := 'MC',
		sArgument2 := '1'
	);	
 	
	fbMcSignalFalingCommand[18](CLK := RxAndTxData.nMcCommandWord_2.7);
	fbMcControlCommandEvents[37](
		bEvent := fbMcSignalFalingCommand[18].Q,
		nEventID := 16#1025,
		sSource := 'Machince Converter Commands',
		sArgument1 := 'MC',
		sArgument2 := '1'
	);
	
	fbMcControlCommandEvents[38](
		bEvent := RxAndTxData.nMcCommandWord_2.8,
		nEventID := 16#1026,
		sSource := 'Machince Converter Commands',
		sArgument1 := 'MC',
		sArgument2 := '1'
	);	
 	
	fbMcSignalFalingCommand[19](CLK := RxAndTxData.nMcCommandWord_2.8);
	fbMcControlCommandEvents[39](
		bEvent := fbMcSignalFalingCommand[19].Q,
		nEventID := 16#1027,
		sSource := 'Machince Converter Commands',
		sArgument1 := 'MC',
		sArgument2 := '1'
	);
	
	fbMcControlCommandEvents[40](
		bEvent := RxAndTxData.nMcCommandWord_2.9,
		nEventID := 16#1028,
		sSource := 'Machince Converter Commands',
		sArgument1 := 'MC',
		sArgument2 := '1'
	);	
 	
	fbMcSignalFalingCommand[20](CLK := RxAndTxData.nMcCommandWord_2.9);
	fbMcControlCommandEvents[41](
		bEvent := fbMcSignalFalingCommand[20].Q,
		nEventID := 16#1029,
		sSource := 'Machince Converter Commands',
		sArgument1 := 'MC',
		sArgument2 := '1'
	);
	
	fbMcControlCommandEvents[42](
		bEvent := RxAndTxData.nMcCommandWord_2.12,
		nEventID := 16#102A,
		sSource := 'Machince Converter Commands',
		sArgument1 := 'MC',
		sArgument2 := '1'
	);	
 	
	fbMcSignalFalingCommand[21](CLK := RxAndTxData.nMcCommandWord_2.12);
	fbMcControlCommandEvents[43](
		bEvent := fbMcSignalFalingCommand[21].Q,
		nEventID := 16#102B,
		sSource := 'Machince Converter Commands',
		sArgument1 := 'MC',
		sArgument2 := '1'
	);
	
	fbMcControlCommandEvents[44](
		bEvent := RxAndTxData.nMcCommandWord_2.13,
		nEventID := 16#102C,
		sSource := 'Machince Converter Commands',
		sArgument1 := 'MC',
		sArgument2 := '1'
	);	
 	
	fbMcSignalFalingCommand[22](CLK := RxAndTxData.nMcCommandWord_2.13);
	fbMcControlCommandEvents[45](
		bEvent := fbMcSignalFalingCommand[22].Q,
		nEventID := 16#102D,
		sSource := 'Machince Converter Commands',
		sArgument1 := 'MC',
		sArgument2 := '1'
	);
	
	fbMcControlCommandEvents[46](
		bEvent := RxAndTxData.nMcCommandWord_2.14,
		nEventID := 16#102E,
		sSource := 'Machince Converter Commands',
		sArgument1 := 'MC',
		sArgument2 := '1'
	);	
 	
	fbMcSignalFalingCommand[23](CLK := RxAndTxData.nMcCommandWord_2.14);
	fbMcControlCommandEvents[47](
		bEvent := fbMcSignalFalingCommand[23].Q,
		nEventID := 16#102F,
		sSource := 'Machince Converter Commands',
		sArgument1 := 'MC',
		sArgument2 := '1'
	);
END_ACTION

ACTION a_McStatusEvents:

(* Events Comming from MC Status *) 

	fbMcStatusEvents[0](
		bEvent := RxAndTxData.nMcStatusWord_1.0,
		nEventID := 16#2000,
		sSource := 'Machince Converter Event',
		sArgument1 := 'MC',
		sArgument2 := '1'
	);	
 	
	fbMcSignalFalingStatus[0](CLK := RxAndTxData.nMcStatusWord_1.0);
	fbMcStatusEvents[1](
		bEvent := fbMcSignalFalingStatus[0].Q,
		nEventID := 16#2001,
		sSource := 'Machince Converter Event',
		sArgument1 := 'MC',
		sArgument2 := '1'
	);
	fbMcStatusEvents[2](
		bEvent := RxAndTxData.nMcStatusWord_1.1,
		nEventID := 16#2002,
		sSource := 'Machince Converter Event',
		sArgument1 := 'MC',
		sArgument2 := '1'
	);	
 	
	fbMcSignalFalingStatus[1](CLK := RxAndTxData.nMcStatusWord_1.1);
	fbMcStatusEvents[3](
		bEvent := fbMcSignalFalingStatus[1].Q,
		nEventID := 16#2003,
		sSource := 'Machince Converter Event',
		sArgument1 := 'MC',
		sArgument2 := '1'
	);
	fbMcStatusEvents[4](
		bEvent := RxAndTxData.nMcStatusWord_1.2,
		nEventID := 16#2004,
		sSource := 'Machince Converter Event',
		sArgument1 := 'MC',
		sArgument2 := '1'
	);	
 	
	fbMcSignalFalingStatus[2](CLK := RxAndTxData.nMcStatusWord_1.2);
	fbMcStatusEvents[5](
		bEvent := fbMcSignalFalingStatus[2].Q,
		nEventID := 16#2005,
		sSource := 'Machince Converter Event',
		sArgument1 := 'MC',
		sArgument2 := '1'
	);
	fbMcStatusEvents[6](
		bEvent := RxAndTxData.nMcStatusWord_1.3,
		nEventID := 16#2006,
		sSource := 'Machince Converter Event',
		sArgument1 := 'MC',
		sArgument2 := '1'
	);	
 	
	fbMcSignalFalingStatus[3](CLK := RxAndTxData.nMcStatusWord_1.3);
	fbMcStatusEvents[7](
		bEvent := fbMcSignalFalingStatus[3].Q,
		nEventID := 16#2007,
		sSource := 'Machince Converter Event',
		sArgument1 := 'MC',
		sArgument2 := '1'
	);
	fbMcStatusEvents[8](
		bEvent := RxAndTxData.nMcStatusWord_1.4,
		nEventID := 16#2008,
		sSource := 'Machince Converter Event',
		sArgument1 := 'MC',
		sArgument2 := '1'
	);	
 	
	fbMcSignalFalingStatus[4](CLK := RxAndTxData.nMcStatusWord_1.4);
	fbMcStatusEvents[9](
		bEvent := fbMcSignalFalingStatus[4].Q,
		nEventID := 16#2009,
		sSource := 'Machince Converter Event',
		sArgument1 := 'MC',
		sArgument2 := '1'
	);
	fbMcStatusEvents[10](
		bEvent := RxAndTxData.nMcStatusWord_1.5,
		nEventID := 16#200A,
		sSource := 'Machince Converter Event',
		sArgument1 := 'MC',
		sArgument2 := '1'
	);	
 	
	fbMcSignalFalingStatus[5](CLK := RxAndTxData.nMcStatusWord_1.5);
	fbMcStatusEvents[11](
		bEvent := fbMcSignalFalingStatus[5].Q,
		nEventID := 16#200B,
		sSource := 'Machince Converter Event',
		sArgument1 := 'MC',
		sArgument2 := '1'
	);
	fbMcStatusEvents[12](
		bEvent := RxAndTxData.nMcStatusWord_1.6,
		nEventID := 16#200C,
		sSource := 'Machince Converter Event',
		sArgument1 := 'MC',
		sArgument2 := '1'
	);	
 	
	fbMcSignalFalingStatus[6](CLK := RxAndTxData.nMcStatusWord_1.6);
	fbMcStatusEvents[13](
		bEvent := fbMcSignalFalingStatus[6].Q,
		nEventID := 16#200D,
		sSource := 'Machince Converter Event',
		sArgument1 := 'MC',
		sArgument2 := '1'
	);
	fbMcStatusEvents[14](
		bEvent := RxAndTxData.nMcStatusWord_1.7,
		nEventID := 16#200E,
		sSource := 'Machince Converter Event',
		sArgument1 := 'MC',
		sArgument2 := '1'
	);	
 	
	fbMcSignalFalingStatus[7](CLK := RxAndTxData.nMcStatusWord_1.7);
	fbMcStatusEvents[15](
		bEvent := fbMcSignalFalingStatus[7].Q,
		nEventID := 16#200F,
		sSource := 'Machince Converter Event',
		sArgument1 := 'MC',
		sArgument2 := '1'
	);
	fbMcStatusEvents[16](
		bEvent := RxAndTxData.nMcStatusWord_1.8,
		nEventID := 16#2010,
		sSource := 'Machince Converter Event',
		sArgument1 := 'MC',
		sArgument2 := '1'
	);	
 	
	fbMcSignalFalingStatus[8](CLK := RxAndTxData.nMcStatusWord_1.8);
	fbMcStatusEvents[17](
		bEvent := fbMcSignalFalingStatus[8].Q,
		nEventID := 16#2011,
		sSource := 'Machince Converter Event',
		sArgument1 := 'MC',
		sArgument2 := '1'
	);
	fbMcStatusEvents[18](
		bEvent := RxAndTxData.nMcStatusWord_1.9,
		nEventID := 16#2012,
		sSource := 'Machince Converter Event',
		sArgument1 := 'MC',
		sArgument2 := '1'
	);	
 	
	fbMcSignalFalingStatus[9](CLK := RxAndTxData.nMcStatusWord_1.9);
	fbMcStatusEvents[19](
		bEvent := fbMcSignalFalingStatus[9].Q,
		nEventID := 16#2013,
		sSource := 'Machince Converter Event',
		sArgument1 := 'MC',
		sArgument2 := '1'
	);
	fbMcStatusEvents[20](
		bEvent := RxAndTxData.nMcStatusWord_1.10,
		nEventID := 16#2014,
		sSource := 'Machince Converter Event',
		sArgument1 := 'MC',
		sArgument2 := '1'
	);	
 	
	fbMcSignalFalingStatus[10](CLK := RxAndTxData.nMcStatusWord_1.10);
	fbMcStatusEvents[21](
		bEvent := fbMcSignalFalingStatus[10].Q,
		nEventID := 16#2015,
		sSource := 'Machince Converter Event',
		sArgument1 := 'MC',
		sArgument2 := '1'
	);
	fbMcStatusEvents[22](
		bEvent := RxAndTxData.nMcStatusWord_1.11,
		nEventID := 16#2016,
		sSource := 'Machince Converter Event',
		sArgument1 := 'MC',
		sArgument2 := '1'
	);	
 	
	fbMcSignalFalingStatus[11](CLK := RxAndTxData.nMcStatusWord_1.11);
	fbMcStatusEvents[23](
		bEvent := fbMcSignalFalingStatus[11].Q,
		nEventID := 16#2017,
		sSource := 'Machince Converter Event',
		sArgument1 := 'MC',
		sArgument2 := '1'
	);
	fbMcStatusEvents[24](
		bEvent := RxAndTxData.nMcStatusWord_1.12,
		nEventID := 16#2018,
		sSource := 'Machince Converter Event',
		sArgument1 := 'MC',
		sArgument2 := '1'
	);	
 	
	fbMcSignalFalingStatus[12](CLK := RxAndTxData.nMcStatusWord_1.12);
	fbMcStatusEvents[25](
		bEvent := fbMcSignalFalingStatus[12].Q,
		nEventID := 16#2019,
		sSource := 'Machince Converter Event',
		sArgument1 := 'MC',
		sArgument2 := '1'
	);
	fbMcStatusEvents[26](
		bEvent := RxAndTxData.nMcStatusWord_1.13,
		nEventID := 16#201A,
		sSource := 'Machince Converter Event',
		sArgument1 := 'MC',
		sArgument2 := '1'
	);	
 	
	fbMcSignalFalingStatus[13](CLK := RxAndTxData.nMcStatusWord_1.13);
	fbMcStatusEvents[27](
		bEvent := fbMcSignalFalingStatus[13].Q,
		nEventID := 16#201B,
		sSource := 'Machince Converter Event',
		sArgument1 := 'MC',
		sArgument2 := '1'
	);
	fbMcStatusEvents[28](
		bEvent := RxAndTxData.nMcStatusWord_1.14,
		nEventID := 16#201C,
		sSource := 'Machince Converter Event',
		sArgument1 := 'MC',
		sArgument2 := '1'
	);	
 	
	fbMcSignalFalingStatus[14](CLK := RxAndTxData.nMcStatusWord_1.14);
	fbMcStatusEvents[29](
		bEvent := fbMcSignalFalingStatus[14].Q,
		nEventID := 16#201D,
		sSource := 'Machince Converter Event',
		sArgument1 := 'MC',
		sArgument2 := '1'
	);
	fbMcStatusEvents[30](
		bEvent := RxAndTxData.nMcStatusWord_2.0,
		nEventID := 16#201E,
		sSource := 'Machince Converter Event',
		sArgument1 := 'MC',
		sArgument2 := '1'
	);	
 	
	fbMcSignalFalingStatus[15](CLK := RxAndTxData.nMcStatusWord_2.0);
	fbMcStatusEvents[31](
		bEvent := fbMcSignalFalingStatus[15].Q,
		nEventID := 16#201F,
		sSource := 'Machince Converter Event',
		sArgument1 := 'MC',
		sArgument2 := '1'
	);
	fbMcStatusEvents[32](
		bEvent := RxAndTxData.nMcStatusWord_2.1,
		nEventID := 16#2020,
		sSource := 'Machince Converter Event',
		sArgument1 := 'MC',
		sArgument2 := '1'
	);	
 	
	fbMcSignalFalingStatus[16](CLK := RxAndTxData.nMcStatusWord_2.1);
	fbMcStatusEvents[33](
		bEvent := fbMcSignalFalingStatus[16].Q,
		nEventID := 16#2021,
		sSource := 'Machince Converter Event',
		sArgument1 := 'MC',
		sArgument2 := '1'
	);
	fbMcStatusEvents[34](
		bEvent := RxAndTxData.nMcStatusWord_2.2,
		nEventID := 16#2022,
		sSource := 'Machince Converter Event',
		sArgument1 := 'MC',
		sArgument2 := '1'
	);	
 	
	fbMcSignalFalingStatus[17](CLK := RxAndTxData.nMcStatusWord_2.2);
	fbMcStatusEvents[35](
		bEvent := fbMcSignalFalingStatus[17].Q,
		nEventID := 16#2023,
		sSource := 'Machince Converter Event',
		sArgument1 := 'MC',
		sArgument2 := '1'
	);
	fbMcStatusEvents[36](
		bEvent := RxAndTxData.nMcStatusWord_2.3,
		nEventID := 16#2024,
		sSource := 'Machince Converter Event',
		sArgument1 := 'MC',
		sArgument2 := '1'
	);	
 	
	fbMcSignalFalingStatus[18](CLK := RxAndTxData.nMcStatusWord_2.3);
	fbMcStatusEvents[37](
		bEvent := fbMcSignalFalingStatus[18].Q,
		nEventID := 16#2025,
		sSource := 'Machince Converter Event',
		sArgument1 := 'MC',
		sArgument2 := '1'
	);
	fbMcStatusEvents[38](
		bEvent := RxAndTxData.nMcStatusWord_2.4,
		nEventID := 16#2026,
		sSource := 'Machince Converter Event',
		sArgument1 := 'MC',
		sArgument2 := '1'
	);	
 	
	fbMcSignalFalingStatus[19](CLK := RxAndTxData.nMcStatusWord_2.4);
	fbMcStatusEvents[39](
		bEvent := fbMcSignalFalingStatus[19].Q,
		nEventID := 16#2027,
		sSource := 'Machince Converter Event',
		sArgument1 := 'MC',
		sArgument2 := '1'
	);
	fbMcStatusEvents[40](
		bEvent := RxAndTxData.nMcStatusWord_2.5,
		nEventID := 16#2028,
		sSource := 'Machince Converter Event',
		sArgument1 := 'MC',
		sArgument2 := '1'
	);	
 	
	fbMcSignalFalingStatus[20](CLK := RxAndTxData.nMcStatusWord_2.5);
	fbMcStatusEvents[41](
		bEvent := fbMcSignalFalingStatus[20].Q,
		nEventID := 16#2029,
		sSource := 'Machince Converter Event',
		sArgument1 := 'MC',
		sArgument2 := '1'
	);
	fbMcStatusEvents[42](
		bEvent := RxAndTxData.nMcStatusWord_2.6,
		nEventID := 16#202A,
		sSource := 'Machince Converter Event',
		sArgument1 := 'MC',
		sArgument2 := '1'
	);	
 	
	fbMcSignalFalingStatus[21](CLK := RxAndTxData.nMcStatusWord_2.6);
	fbMcStatusEvents[43](
		bEvent := fbMcSignalFalingStatus[21].Q,
		nEventID := 16#202B,
		sSource := 'Machince Converter Event',
		sArgument1 := 'MC',
		sArgument2 := '1'
	);
	fbMcStatusEvents[44](
		bEvent := RxAndTxData.nMcStatusWord_2.7,
		nEventID := 16#202C,
		sSource := 'Machince Converter Event',
		sArgument1 := 'MC',
		sArgument2 := '1'
	);	
 	
	fbMcSignalFalingStatus[22](CLK := RxAndTxData.nMcStatusWord_2.7);
	fbMcStatusEvents[45](
		bEvent := fbMcSignalFalingStatus[22].Q,
		nEventID := 16#202D,
		sSource := 'Machince Converter Event',
		sArgument1 := 'MC',
		sArgument2 := '1'
	);
	fbMcStatusEvents[46](
		bEvent := RxAndTxData.nMcStatusWord_2.8,
		nEventID := 16#202E,
		sSource := 'Machince Converter Event',
		sArgument1 := 'MC',
		sArgument2 := '1'
	);	
 	
	fbMcSignalFalingStatus[23](CLK := RxAndTxData.nMcStatusWord_2.8);
	fbMcStatusEvents[47](
		bEvent := fbMcSignalFalingStatus[23].Q,
		nEventID := 16#202F,
		sSource := 'Machince Converter Event',
		sArgument1 := 'MC',
		sArgument2 := '1'
	);
	fbMcStatusEvents[48](
		bEvent := RxAndTxData.nMcStatusWord_2.9,
		nEventID := 16#2030,
		sSource := 'Machince Converter Event',
		sArgument1 := 'MC',
		sArgument2 := '1'
	);	
 	
	fbMcSignalFalingStatus[24](CLK := RxAndTxData.nMcStatusWord_2.9);
	fbMcStatusEvents[49](
		bEvent := fbMcSignalFalingStatus[24].Q,
		nEventID := 16#2031,
		sSource := 'Machince Converter Event',
		sArgument1 := 'MC',
		sArgument2 := '1'
	);
	fbMcStatusEvents[50](
		bEvent := RxAndTxData.nMcStatusWord_2.10,
		nEventID := 16#2032,
		sSource := 'Machince Converter Event',
		sArgument1 := 'MC',
		sArgument2 := '1'
	);	
 	
	fbMcSignalFalingStatus[25](CLK := RxAndTxData.nMcStatusWord_2.10);
	fbMcStatusEvents[51](
		bEvent := fbMcSignalFalingStatus[25].Q,
		nEventID := 16#2033,
		sSource := 'Machince Converter Event',
		sArgument1 := 'MC',
		sArgument2 := '1'
	);
	fbMcStatusEvents[52](
		bEvent := RxAndTxData.nMcStatusWord_2.11,
		nEventID := 16#2034,
		sSource := 'Machince Converter Event',
		sArgument1 := 'MC',
		sArgument2 := '1'
	);	
 	
	fbMcSignalFalingStatus[26](CLK := RxAndTxData.nMcStatusWord_2.11);
	fbMcStatusEvents[53](
		bEvent := fbMcSignalFalingStatus[26].Q,
		nEventID := 16#2035,
		sSource := 'Machince Converter Event',
		sArgument1 := 'MC',
		sArgument2 := '1'
	);
	fbMcStatusEvents[54](
		bEvent := RxAndTxData.nMcStatusWord_2.12,
		nEventID := 16#2036,
		sSource := 'Machince Converter Event',
		sArgument1 := 'MC',
		sArgument2 := '1'
	);	
 	
	fbMcSignalFalingStatus[27](CLK := RxAndTxData.nMcStatusWord_2.12);
	fbMcStatusEvents[55](
		bEvent := fbMcSignalFalingStatus[27].Q,
		nEventID := 16#2037,
		sSource := 'Machince Converter Event',
		sArgument1 := 'MC',
		sArgument2 := '1'
	);
	fbMcStatusEvents[56](
		bEvent := RxAndTxData.nMcStatusWord_2.13,
		nEventID := 16#2038,
		sSource := 'Machince Converter Event',
		sArgument1 := 'MC',
		sArgument2 := '1'
	);	
 	
	fbMcSignalFalingStatus[28](CLK := RxAndTxData.nMcStatusWord_2.13);
	fbMcStatusEvents[57](
		bEvent := fbMcSignalFalingStatus[28].Q,
		nEventID := 16#2039,
		sSource := 'Machince Converter Event',
		sArgument1 := 'MC',
		sArgument2 := '1'
	);
	fbMcStatusEvents[58](
		bEvent := RxAndTxData.nMcStatusWord_2.14,
		nEventID := 16#203A,
		sSource := 'Machince Converter Event',
		sArgument1 := 'MC',
		sArgument2 := '1'
	);	
 	
	fbMcSignalFalingStatus[29](CLK := RxAndTxData.nMcStatusWord_2.14);
	fbMcStatusEvents[59](
		bEvent := fbMcSignalFalingStatus[29].Q,
		nEventID := 16#203B,
		sSource := 'Machince Converter Event',
		sArgument1 := 'MC',
		sArgument2 := '1'
	);
	fbMcStatusEvents[60](
		bEvent := RxAndTxData.nMcStatusWord_2.15,
		nEventID := 16#203C,
		sSource := 'Machince Converter Event',
		sArgument1 := 'MC',
		sArgument2 := '1'
	);	
 	
	fbMcSignalFalingStatus[30](CLK := RxAndTxData.nMcStatusWord_2.16);
	fbMcStatusEvents[61](
		bEvent := fbMcSignalFalingStatus[30].Q,
		nEventID := 16#203D,
		sSource := 'Machince Converter Event',
		sArgument1 := 'MC',
		sArgument2 := '1'
	);
END_ACTION

END_PROGRAM

// ---- EventLogger/FunctionBlocks/FB_EventMessage.TcPOU
FUNCTION_BLOCK FB_EventMessage
VAR_INPUT
    bEvent            : BOOL;
    nEventID         : UDINT;
    sSource            : STRING;
    sArgument1        : STRING;
    sArgument2        : STRING;
    
END_VAR
VAR_OUTPUT
END_VAR
VAR
    bIsInitialized     : BOOL;
    
    fbSourceInfo    : FB_TcSourceInfo;
    fbMessage         : FB_TcMessage;
    eventEntry        : TcEventEntry;
    fbRtEvent        : R_TRIG;
    
    hr                 : HRESULT;
    hrLastError        : HRESULT;
END_VAR


(* Initialization *)
    IF NOT bIsInitialized THEN
        bIsInitialized := TRUE;
    (* This part is used to change events class depending on the ivent ID for example for Warning or for Info *)
    IF nEventID < 16#2000 THEN
        eventEntry := Tc_Events.ConvCommandEvents.CmdUnlockRamp_1;         // Converter Commands
    ELSIF nEventID < 16#3000 THEN
        eventEntry := Tc_Events.StatusWordEvents.StateOn_1;             // Converter Status Events
    END_IF
        eventEntry.nEventId := nEventID;
        fbSourceInfo.Clear();
        fbSourceInfo.sName := sSource;
        hr := fbMessage.CreateEx(eventEntry, ipSourceInfo := fbSourceInfo);
    END_IF
    
    IF FAILED(hr) THEN
        hrLastError := hr;
    END_IF 
    
    fbMessage.ipArguments.Clear().AddString(sArgument1).AddString(sArgument2);
    
(* event trigger *)
    fbRtEvent(CLK := bEvent);
    
(* send message *)
    IF fbRtEvent.Q THEN
        hr := fbMessage.Send(0);
        UtilityVariables.nEventsInEventLogger := UtilityVariables.nEventsInEventLogger + 1; // Counts the nuber of events stored in PLC ceche
        IF FAILED(hr) THEN
            hrLastError := hr;
        END_IF
    END_IF

END_FUNCTION_BLOCK

// ---- EventLogger/FunctionBlocks/Common/P_Timer.TcPOU
PROGRAM P_Timer
VAR
    fbSystemTime             : FB_LocalSystemTime;
    dtCurrentDateTime        : DT;
    sCurrentDateTime         : STRING;
    sDateTime                : STRING;
    bSecond                  : BOOL;
    nSecond                  : WORD;
    bPulsels                 : BOOL;
    bPulse05s                : BOOL;
    
    fbRtSecond               : R_TRIG;
    fbLow_1s                 : TON;
    fbHigh_1s                : TOF;
    fbLow_05s                : TON;
    fbHigh_05s               : TOF;
    
    
    
    fbSystemTimefbSystemTime: INT;
END_VAR

(* Synchronize system time *)

    fbSystemTime(
        bEnable  := TRUE, 
        dwCycle  := 5 , 
        dwOpt    := 1 , 
    );
    
    dtCurrentDateTime   := SYSTEMTIME_TO_DT(fbSystemTime.systemTime);
    sCurrentDateTime    := MID(DT_TO_STRING(dtCurrentDateTime), 19, 4);
    
(* Convert timetamp because ':' ivalid if file vame *)

    sDateTime := sCurrentDateTime;
    sDateTIme := replace(sDateTime, '-', 1, 11);
    sDateTIme := replace(sDateTime, '-', 1, 14);
    sDateTIme := replace(sDateTime, '-', 1, 17);
    
(* 1 sek. trigger *)
    
    fbRtSecond( CLK := fbSystemTime.systemTime.wSecond <> nSecond, Q => bSecond);
    nSecond := fbSystemTime.systemTime.wSecond;
    
(* 1 sek. blinking puls *)
    
    fbLow_1s(IN := NOT bPulsels, PT := T#500MS);
    fbHigh_1s(IN := fbLow_1s.Q, PT := T#500MS, Q => bPulsels);
    
(* 0.5 sek. blinking puls *)
    
    fbLow_05s(IN := NOT bPulse05s, PT := T#150MS);
    fbHigh_05s(IN := fbLow_05s.Q, PT := T#150MS, Q => bPulse05s);

END_PROGRAM

// ---- DUTs/FB_GetFaultWordsFromProtxConverter.TcPOU
FUNCTION_BLOCK FB_GetFaultWordsFromProtxConverter
VAR_INPUT
    stOutputVectorInteger : ST_OutputVectorInteger1;
    stOutputVectorReal : ST_OutputVectorReal1;
END_VAR
VAR
    stLcFaultWord1 : ST_LcFaultWord1;
    stLcFaultWord2 : ST_LcFaultWord2;
    stLcFaultWord3 : ST_LcFaultWord3;
    stLcFaultWord4 : ST_LcFaultWord4;
    stMcFaultWord1 : ST_McFaultWord1;
    stMcFaultWord2 : ST_McFaultWord2;
    stMcFaultWord3 : ST_McFaultWord3;
    stMcFaultWord4 : ST_McFaultWord4;
    
    wLcFaultWord1     : WORD;
     wLcFaultWord2     : WORD;
    wLcFaultWord3     : WORD;
    wLcFaultWord4     : WORD;
    wMcFaultWord1     : WORD;
     wMcFaultWord2     : WORD;
    wMcFaultWord3     : WORD;
    wMcFaultWord4     : WORD;


    nLcFaultWord1     : LINT;
     nLcFaultWord2     : LINT;
    nLcFaultWord3     : LINT;
    nLcFaultWord4     : LINT;
    nMcFaultWord1     : LINT;
     nMcFaultWord2     : LINT;
    nMcFaultWord3     : LINT;
    nMcFaultWord4     : LINT;
    
    
     
END_VAR

/// Conversion from LINT to WORD {{{
wLcFaultWord1 := TO_WORD(TO_INT(stOutputVectorInteger.Element02_LcDriveFaultCategoryB));
wLcFaultWord2 := TO_WORD(TO_INT(stOutputVectorInteger.Element03_LcDriveFaultCategoryC));
wLcFaultWord3 := TO_WORD(TO_INT(stOutputVectorInteger.Element04_LcDriveFaultCategoryC));
wLcFaultWord4 := TO_WORD(TO_INT(stOutputVectorInteger.Element05_LcDriveFaultCategoryD));
wMcFaultWord1 := TO_WORD(TO_INT(stOutputVectorInteger.Element14_McDriveFaultCategoryB));
wMcFaultWord2 := TO_WORD(TO_INT(stOutputVectorInteger.Element15_McDriveFaultCategoryC));
wMcFaultWord3 := TO_WORD(TO_INT(stOutputVectorInteger.Element16_McDriveFaultCategoryC));
wMcFaultWord4 := TO_WORD(TO_INT(stOutputVectorInteger.Element17_McDriveFaultCategoryD));
///}}}

/// LC Fault Word 1 {{{
RxAndTxData.stLcFaultWord1.Bit00_FaultInputAryEcat := wLcFaultWord1.0;
RxAndTxData.stLcFaultWord1.Bit01_FPGA := wLcFaultWord1.1;
RxAndTxData.stLcFaultWord1.Bit02_Watchdog := wLcFaultWord1.2;
RxAndTxData.stLcFaultWord1.Bit03_UdcMax := wLcFaultWord1.3;
RxAndTxData.stLcFaultWord1.Bit08_UceFault := wLcFaultWord1.8;
///}}} 
    
/// LC Fault Word 2 {{{
RxAndTxData.stLcFaultWord2.Bit00_PibSupply := wLcFaultWord2.0;
RxAndTxData.stLcFaultWord2.Bit01_MeasurementConnectorLoop := wLcFaultWord2.1;
RxAndTxData.stLcFaultWord2.Bit02_FaultLoop := wLcFaultWord2.2;
RxAndTxData.stLcFaultWord2.Bit03_AmplifierConnector := wLcFaultWord2.3;
RxAndTxData.stLcFaultWord2.Bit04_TermSupply := wLcFaultWord2.4;
RxAndTxData.stLcFaultWord2.Bit05_Overcurrent := wLcFaultWord2.5;
RxAndTxData.stLcFaultWord2.Bit06_ShortCircuit := wLcFaultWord2.6;
RxAndTxData.stLcFaultWord2.Bit07_DcConnection := wLcFaultWord2.7;
RxAndTxData.stLcFaultWord2.Bit08_ThHSMax := wLcFaultWord2.8;
RxAndTxData.stLcFaultWord2.Bit09_ShortCircuit24V := wLcFaultWord2.9;
RxAndTxData.stLcFaultWord2.Bit10_FieldBus := wLcFaultWord2.10;
RxAndTxData.stLcFaultWord2.Bit11_FLinkRxMc := wLcFaultWord2.11;
RxAndTxData.stLcFaultWord2.Bit12_EarthFault := wLcFaultWord2.12;
RxAndTxData.stLcFaultWord2.Bit13_UdcMin := wLcFaultWord2.13;
RxAndTxData.stLcFaultWord2.Bit15_ExtFault := wLcFaultWord2.15;
///}}}
    
/// LC Fault Word 3 {{{
RxAndTxData.stLcFaultWord3.Bit00_ULineVoltage := wLcFaultWord3.0;
RxAndTxData.stLcFaultWord3.Bit01_ULineMeasurement := wLcFaultWord3.1;
RxAndTxData.stLcFaultWord3.Bit02_AcFuse := wLcFaultWord3.2;
RxAndTxData.stLcFaultWord3.Bit03_FbLineContactor := wLcFaultWord3.3;
RxAndTxData.stLcFaultWord3.Bit04_Charging := wLcFaultWord3.4;
RxAndTxData.stLcFaultWord3.Bit05_LineFilter := wLcFaultWord3.5;
///}}}

/// LC Fault Word 4 {{{
RxAndTxData.stLcFaultWord4.Bit00_NTC := wLcFaultWord4.0;
RxAndTxData.stLcFaultWord4.Bit01_ThHsMin := wLcFaultWord4.1;
RxAndTxData.stLcFaultWord4.Bit02_CoolingSystem := wLcFaultWord4.2;
RxAndTxData.stLcFaultWord4.Bit03_ControllerCabinetFan := wLcFaultWord4.3;
RxAndTxData.stLcFaultWord4.Bit04_ConverterCubiceOvertemp := wLcFaultWord4.4;
RxAndTxData.stLcFaultWord4.Bit05_CubicleAuxSupply := wLcFaultWord4.5;
RxAndTxData.stLcFaultWord4.Bit09_FeedInCubicleOvertemp := wLcFaultWord4.9;
RxAndTxData.stLcFaultWord4.Bit10_TrafoOvertemp := wLcFaultWord4.10;
RxAndTxData.stLcFaultWord4.Bit11_Isolation := wLcFaultWord4.11;
///}}}

/// MC Fault Word 1 {{{
RxAndTxData.stMcFaultWord1.Bit00_FaultInputAryEcat := wMcFaultWord1.0;
RxAndTxData.stMcFaultWord1.Bit01_FPGA := wMcFaultWord1.1;
RxAndTxData.stMcFaultWord1.Bit02_Watchdog := wMcFaultWord1.2;
RxAndTxData.stMcFaultWord1.Bit03_UdcMax := wMcFaultWord1.3;
RxAndTxData.stMcFaultWord1.Bit08_UceFault := wMcFaultWord1.8;
///}}}

/// MC Fault Word 2 {{{
RxAndTxData.stMcFaultWord2.Bit00_PibSupply := wMcFaultWord2.0;
RxAndTxData.stMcFaultWord2.Bit01_MeasurementConnectorLoop := wMcFaultWord2.1;
RxAndTxData.stMcFaultWord2.Bit02_FaultLoop := wMcFaultWord2.2;
RxAndTxData.stMcFaultWord2.Bit03_AmplifierConnector := wMcFaultWord2.3;
RxAndTxData.stMcFaultWord2.Bit04_TermSupply := wMcFaultWord2.4;
RxAndTxData.stMcFaultWord2.Bit05_Overcurrent := wMcFaultWord2.5;
RxAndTxData.stMcFaultWord2.Bit06_ShortCircuit := wMcFaultWord2.6;
RxAndTxData.stMcFaultWord2.Bit07_DcConnection := wMcFaultWord2.7;
RxAndTxData.stMcFaultWord2.Bit08_ThHSMax := wMcFaultWord2.8;
RxAndTxData.stMcFaultWord2.Bit09_ShortCircuit24V := wMcFaultWord2.9;
RxAndTxData.stMcFaultWord2.Bit10_FieldBus := wMcFaultWord2.10;
RxAndTxData.stMcFaultWord2.Bit11_FLinkRxMc := wMcFaultWord2.11;
RxAndTxData.stMcFaultWord2.Bit12_EarthFault := wMcFaultWord2.12;
RxAndTxData.stMcFaultWord2.Bit13_UdcMin := wMcFaultWord2.13;
RxAndTxData.stMcFaultWord2.Bit15_ExtFault := wMcFaultWord2.15;
///}}}

/// MC Fault Word 3 {{{
RxAndTxData.stMcFaultWord3.Bit00_EncoderFault := wMcFaultWord3.0;
RxAndTxData.stMcFaultWord3.Bit01_BlockFault := wMcFaultWord3.1;
RxAndTxData.stMcFaultWord3.Bit02_OverspeedFault := wMcFaultWord3.2;
RxAndTxData.stMcFaultWord3.Bit03_BrakeFault := wMcFaultWord3.3;
RxAndTxData.stMcFaultWord3.Bit04_InterlockRotating := wMcFaultWord3.4;
RxAndTxData.stMcFaultWord3.Bit05_DcOutputSwitches := wMcFaultWord3.5;
RxAndTxData.stMcFaultWord3.Bit06_DcOutputOfRange := wMcFaultWord3.6;
RxAndTxData.stMcFaultWord3.Bit07_DcSwitchOnSequence := wMcFaultWord3.7;
///}}}

/// MC Fault Word 4 {{{
RxAndTxData.stMcFaultWord4.Bit00_NTC := wMcFaultWord4.0;
RxAndTxData.stMcFaultWord4.Bit01_ThHsMin := wMcFaultWord4.1;
RxAndTxData.stMcFaultWord4.Bit03_ControllerCabinetFan := wMcFaultWord4.3;
RxAndTxData.stMcFaultWord4.Bit04_ConverterCubiceOvertemp := wMcFaultWord4.4;
RxAndTxData.stMcFaultWord4.Bit05_CubicleAuxSupply := wMcFaultWord4.5;
RxAndTxData.stMcFaultWord4.Bit06_MotorTemp := wMcFaultWord4.6;
RxAndTxData.stMcFaultWord4.Bit08_FrequLock := wMcFaultWord4.8;
RxAndTxData.stMcFaultWord4.Bit09_ConverterOverload := wMcFaultWord4.9;
///}}}

END_FUNCTION_BLOCK

// ---- DUTs/FB_PrepareInputVectorsFromProTxCovnerter.TcPOU
FUNCTION_BLOCK FB_PrepareInputVectorsFromProTxCovnerter
VAR_INPUT
END_VAR
VAR_OUTPUT
END_VAR
VAR
	wLcStatusWord_1 				: WORD;
	wLcStatusWord_2					: WORD;
	wMcStatusWord_1 				: WORD;
	wMcStatusWord_2					: WORD;
	wLcFaultWord1					: WORD; // write description
	wLcFaultWord2					: WORD;
	wLcFaultWord3					: WORD;
	wLcFaultWord4					: WORD;
	wMcFaultWord1					: WORD;
	wMcFaultWord2					: WORD;
	wMcFaultWord3					: WORD;
	wMcFaultWord4					: WORD;
END_VAR

/// Converting Integer Inputs from UDINT to Word {{{
	wLcStatusWord_1 := TO_WORD(RxAndTxData.nLcStatusWord_1);
	wLcStatusWord_2 := TO_WORD(RxAndTxData.nLcStatusWord_2);
	wMcStatusWord_1 := TO_WORD(RxAndTxData.nMcStatusWord_1);
	wMcStatusWord_2 := TO_WORD(RxAndTxData.nMcStatusWord_2);
	
///}}}

/// Converting the LC Status Word 1 from UDINT to Structure {{{
	StatusAndCommandWordsStructures.stLcStatusWord_1.Bit00_StateReady 				:= wLcStatusWord_1.0;
	StatusAndCommandWordsStructures.stLcStatusWord_1.Bit01_StateOn 					:= wLcStatusWord_1.1;
	StatusAndCommandWordsStructures.stLcStatusWord_1.Bit02_CtrlRun 					:= wLcStatusWord_1.2;
	StatusAndCommandWordsStructures.stLcStatusWord_1.Bit03_CollFault 				:= wLcStatusWord_1.3;
	StatusAndCommandWordsStructures.stLcStatusWord_1.Bit04_DriveReleaseActive 		:= wLcStatusWord_1.4;
	StatusAndCommandWordsStructures.stLcStatusWord_1.Bit05_StatePowerOk 			:= wLcStatusWord_1.5;
	StatusAndCommandWordsStructures.stLcStatusWord_1.Bit06_StateDisable 			:= wLcStatusWord_1.6;
	StatusAndCommandWordsStructures.stLcStatusWord_1.Bit07_Warning 					:= wLcStatusWord_1.7;
	StatusAndCommandWordsStructures.stLcStatusWord_1.Bit08_PhaseLoss 				:= wLcStatusWord_1.8;
	StatusAndCommandWordsStructures.stLcStatusWord_1.Bit09_BusSelected 				:= wLcStatusWord_1.9;
	StatusAndCommandWordsStructures.stLcStatusWord_1.Bit10_uu 						:= wLcStatusWord_1.10;
	StatusAndCommandWordsStructures.stLcStatusWord_1.Bit11_uu 						:= wLcStatusWord_1.11;
	StatusAndCommandWordsStructures.stLcStatusWord_1.Bit12_ReleaseMc 				:= wLcStatusWord_1.12;
	StatusAndCommandWordsStructures.stLcStatusWord_1.Bit13_StateTestModeOn 			:= wLcStatusWord_1.13;
	StatusAndCommandWordsStructures.stLcStatusWord_1.Bit14_InternalAliveToggle 		:= wLcStatusWord_1.14;
	StatusAndCommandWordsStructures.stLcStatusWord_1.Bit15_MainAliveToggle 			:= wLcStatusWord_1.15;
///}}}

/// Converting the LC Status Word 2 from UDINT to Structure {{{
	StatusAndCommandWordsStructures.stLcStatusWord_2.Bit00_FaultB					:= wLcStatusWord_2.0;
	StatusAndCommandWordsStructures.stLcStatusWord_2.Bit01_FaultC					:= wLcStatusWord_2.1;
	StatusAndCommandWordsStructures.stLcStatusWord_2.Bit02_FaultC 					:= wLcStatusWord_2.2;
	StatusAndCommandWordsStructures.stLcStatusWord_2.Bit03_FaultDWarning 			:= wLcStatusWord_2.3;
	StatusAndCommandWordsStructures.stLcStatusWord_2.Bit04_TrafoOvertempWarning		:= wLcStatusWord_2.4;
	StatusAndCommandWordsStructures.stLcStatusWord_2.Bit05_TrafoInsolationWarning	:= wLcStatusWord_2.5;
	StatusAndCommandWordsStructures.stLcStatusWord_2.Bit06_uu						:= wLcStatusWord_2.6;
	StatusAndCommandWordsStructures.stLcStatusWord_2.Bit07_uu						:= wLcStatusWord_2.7;
	StatusAndCommandWordsStructures.stLcStatusWord_2.Bit08_uu						:= wLcStatusWord_2.8;
	StatusAndCommandWordsStructures.stLcStatusWord_2.Bit09_uu						:= wLcStatusWord_2.9;
	StatusAndCommandWordsStructures.stLcStatusWord_2.Bit10_ThHSWarning				:= wLcStatusWord_2.10;
	StatusAndCommandWordsStructures.stLcStatusWord_2.Bit11_ThHSMaxWarning			:= wLcStatusWord_2.11;
	StatusAndCommandWordsStructures.stLcStatusWord_2.Bit12_ParSetBit00				:= wLcStatusWord_2.12;
	StatusAndCommandWordsStructures.stLcStatusWord_2.Bit13_ParSetBit01				:= wLcStatusWord_2.13;
	StatusAndCommandWordsStructures.stLcStatusWord_2.Bit14_ParSetBit02				:= wLcStatusWord_2.14;
	StatusAndCommandWordsStructures.stLcStatusWord_2.Bit15_ParSetBit03				:= wLcStatusWord_2.15;
///}}}

/// Converting the MC Status Word 1 from UDINT to Structure {{{
	StatusAndCommandWordsStructures.stMcStatusWord_1.Bit00_StateReady 				:= wMcStatusWord_1.0;
	StatusAndCommandWordsStructures.stMcStatusWord_1.Bit01_StateOn  				:= wMcStatusWord_1.1;
	StatusAndCommandWordsStructures.stMcStatusWord_1.Bit02_CtrlRun  				:= wMcStatusWord_1.2;
	StatusAndCommandWordsStructures.stMcStatusWord_1.Bit03_CollFault  				:= wMcStatusWord_1.3;
	StatusAndCommandWordsStructures.stMcStatusWord_1.Bit04_DriveReleaseActive  		:= wMcStatusWord_1.4;
	StatusAndCommandWordsStructures.stMcStatusWord_1.Bit05_StateFastStop  			:= wMcStatusWord_1.5;
	StatusAndCommandWordsStructures.stMcStatusWord_1.Bit06_StateDisable	 			:= wMcStatusWord_1.6;
	StatusAndCommandWordsStructures.stMcStatusWord_1.Bit07_Warning  				:= wMcStatusWord_1.7;
	StatusAndCommandWordsStructures.stMcStatusWord_1.Bit08_SpeedCtrlLimited	 		:= wMcStatusWord_1.8;
	StatusAndCommandWordsStructures.stMcStatusWord_1.Bit09_BusSelected  			:= wMcStatusWord_1.9;
	StatusAndCommandWordsStructures.stMcStatusWord_1.Bit10_XnIsEqualToWn  			:= wMcStatusWord_1.10;
	StatusAndCommandWordsStructures.stMcStatusWord_1.Bit11_WiqTLimited  			:= wMcStatusWord_1.11;
	StatusAndCommandWordsStructures.stMcStatusWord_1.Bit12_XnIsEqualToZero  		:= wMcStatusWord_1.12;
	StatusAndCommandWordsStructures.stMcStatusWord_1.Bit13_NCtrlenable  			:= wMcStatusWord_1.13;
	StatusAndCommandWordsStructures.stMcStatusWord_1.Bit14_ExtrnalTorqueRelease  	:= wMcStatusWord_1.14;
	StatusAndCommandWordsStructures.stMcStatusWord_1.Bit15_MainAliveToggle  		:= wMcStatusWord_1.15;
///}}}

/// Converting the MC Status Word 2 from UDINT to Structure {{{
	StatusAndCommandWordsStructures.stMcStatusWord_2.Bit00_FaultB 					:= wMcStatusWord_2.0;
	StatusAndCommandWordsStructures.stMcStatusWord_2.Bit01_FaultC 					:= wMcStatusWord_2.1;
	StatusAndCommandWordsStructures.stMcStatusWord_2.Bit02_FaultC 					:= wMcStatusWord_2.2;
	StatusAndCommandWordsStructures.stMcStatusWord_2.Bit03_FaultDWarning 			:= wMcStatusWord_2.3;
	StatusAndCommandWordsStructures.stMcStatusWord_2.Bit04_MRegActive 				:= wMcStatusWord_2.4;
	StatusAndCommandWordsStructures.stMcStatusWord_2.Bit05_torqueRegEnable 			:= wMcStatusWord_2.5;
	StatusAndCommandWordsStructures.stMcStatusWord_2.Bit06_ConverterI2tLinitWarning := wMcStatusWord_2.6;
	StatusAndCommandWordsStructures.stMcStatusWord_2.Bit07_ConverterI2tLinitActive 	:= wMcStatusWord_2.7;
	StatusAndCommandWordsStructures.stMcStatusWord_2.Bit08_MotorI2tLinitWarning 	:= wMcStatusWord_2.8;
	StatusAndCommandWordsStructures.stMcStatusWord_2.Bit09_MotorI2tLinitActive 		:= wMcStatusWord_2.9;
	StatusAndCommandWordsStructures.stMcStatusWord_2.Bit10_ThHSWarning 				:= wMcStatusWord_2.10;
	StatusAndCommandWordsStructures.stMcStatusWord_2.Bit11_ThHSMaxWarning 			:= wMcStatusWord_2.11;
	StatusAndCommandWordsStructures.stMcStatusWord_2.Bit12_windingTempWarning 		:= wMcStatusWord_2.12;
	StatusAndCommandWordsStructures.stMcStatusWord_2.Bit13_BearingTempWarning 		:= wMcStatusWord_2.13;
	StatusAndCommandWordsStructures.stMcStatusWord_2.Bit14_Forward 					:= wMcStatusWord_2.14;
	StatusAndCommandWordsStructures.stMcStatusWord_2.Bit15_Reverse 					:= wMcStatusWord_2.15;
///}}}

/// Writing Output Real Vector Into the Structure {{{
	
///}}}

END_FUNCTION_BLOCK

// ---- DUTs/FB_GetStatusWordsFromProTxConverter.TcPOU
FUNCTION_BLOCK FB_GetStatusWordsFromProTxConverter
VAR_INPUT
    stOutputVectorInteger : ST_OutputVectorInteger1;
    stOutputVectorReal : ST_OutputVectorReal1;
END_VAR
VAR
    stLcMainStatusWord : ST_LcStatusWord_1_ProfiDrive;
    stMcMainStatusWord : ST_McStatusWord_1_ProfiDrive;
    stLcAuxiliaryStatusWord : ST_LcStatusWord_2_ProfiDrive;
    stMcAuxiliaryStatusWord : ST_LcStatusWord_2_ProfiDrive;
    
    wLcMainStatusWord : WORD;
    wMcMainStatusWord : WORD;
    wLcAuxiliaryStatusWord : WORD;
    wMcAuxiliaryStatusWord : WORD;
END_VAR

wLcMainStatusWord := TO_WORD(TO_INT(stOutputVectorInteger.Element00_LcMainStatusWord));
wMcMainStatusWord := TO_WORD(TO_INT(stOutputVectorInteger.Element01_LcAuxiliaryStatusWord));
wLcAuxiliaryStatusWord := TO_WORD(TO_INT(stOutputVectorInteger.Element12_McMainStatusWord));
wMcAuxiliaryStatusWord := TO_WORD(TO_INT(stOutputVectorInteger.Element13_McAuxiliaryStatusWord));

/// Copyng LC Main Status Word Into Structure {{{
RxAndTxData.stLcMainStatusWord.Bit00_StateReady := wLcMainStatusWord.0;
RxAndTxData.stLcMainStatusWord.Bit01_StateOn := wLcMainStatusWord.1;
RxAndTxData.stLcMainStatusWord.Bit02_CtrlRun := wLcMainStatusWord.2;
RxAndTxData.stLcMainStatusWord.Bit03_CollFault := wLcMainStatusWord.3;
RxAndTxData.stLcMainStatusWord.Bit04_DriveReleaseActive := wLcMainStatusWord.4;
RxAndTxData.stLcMainStatusWord.Bit05_StatePowerOk := wLcMainStatusWord.5;
RxAndTxData.stLcMainStatusWord.Bit06_StateDisable := wLcMainStatusWord.6;
RxAndTxData.stLcMainStatusWord.Bit07_Warning := wLcMainStatusWord.7;
RxAndTxData.stLcMainStatusWord.Bit08_PhaseLoss := wLcMainStatusWord.8;
RxAndTxData.stLcMainStatusWord.Bit09_BusSelected := wLcMainStatusWord.9;
RxAndTxData.stLcMainStatusWord.Bit10_uu := wLcMainStatusWord.10;
RxAndTxData.stLcMainStatusWord.Bit11_uu := wLcMainStatusWord.11;
RxAndTxData.stLcMainStatusWord.Bit12_ReleaseMc := wLcMainStatusWord.12;
RxAndTxData.stLcMainStatusWord.Bit13_StateTestModeOn := wLcMainStatusWord.13;
RxAndTxData.stLcMainStatusWord.Bit14_InternalAliveToggle := wLcMainStatusWord.14;
RxAndTxData.stLcMainStatusWord.Bit15_MainAliveToggle := wLcMainStatusWord.15;
///}}}

/// Copyng LC Auxiliary Status Word Into Structure {{{
RxAndTxData.stLcAuxiliaryStatusWord.Bit00_FaultB := wLcAuxiliaryStatusWord.0;
RxAndTxData.stLcAuxiliaryStatusWord.Bit01_FaultC := wLcAuxiliaryStatusWord.1;
RxAndTxData.stLcAuxiliaryStatusWord.Bit02_FaultC := wLcAuxiliaryStatusWord.2;
RxAndTxData.stLcAuxiliaryStatusWord.Bit03_FaultDWarning := wLcAuxiliaryStatusWord.3;
RxAndTxData.stLcAuxiliaryStatusWord.Bit04_TrafoOvertempWarning := wLcAuxiliaryStatusWord.4;
RxAndTxData.stLcAuxiliaryStatusWord.Bit05_TrafoInsolationWarning := wLcAuxiliaryStatusWord.5;
RxAndTxData.stLcAuxiliaryStatusWord.Bit06_uu := wLcAuxiliaryStatusWord.6;
RxAndTxData.stLcAuxiliaryStatusWord.Bit07_uu := wLcAuxiliaryStatusWord.7;
RxAndTxData.stLcAuxiliaryStatusWord.Bit08_uu := wLcAuxiliaryStatusWord.8;
RxAndTxData.stLcAuxiliaryStatusWord.Bit09_uu := wLcAuxiliaryStatusWord.9;
RxAndTxData.stLcAuxiliaryStatusWord.Bit10_ThHSWarning := wLcAuxiliaryStatusWord.10;
RxAndTxData.stLcAuxiliaryStatusWord.Bit11_ThHSMaxWarning := wLcAuxiliaryStatusWord.11;
RxAndTxData.stLcAuxiliaryStatusWord.Bit12_ParSetBit00 := wLcAuxiliaryStatusWord.12;
RxAndTxData.stLcAuxiliaryStatusWord.Bit13_ParSetBit01 := wLcAuxiliaryStatusWord.13;
RxAndTxData.stLcAuxiliaryStatusWord.Bit14_ParSetBit02 := wLcAuxiliaryStatusWord.14;
RxAndTxData.stLcAuxiliaryStatusWord.Bit15_ParSetBit03 := wLcAuxiliaryStatusWord.15;    
///}}}

/// Copyng MC Main Status Word Into Structure {{{
RxAndTxData.stMcMainStatusWord.Bit00_StateReady := wMcMainStatusWord.0;
RxAndTxData.stMcMainStatusWord.Bit01_StateOn := wMcMainStatusWord.1;
RxAndTxData.stMcMainStatusWord.Bit02_CtrlRun := wMcMainStatusWord.2;
RxAndTxData.stMcMainStatusWord.Bit03_CollFault := wMcMainStatusWord.3;
RxAndTxData.stMcMainStatusWord.Bit04_DriveReleaseActive := wMcMainStatusWord.4;
RxAndTxData.stMcMainStatusWord.Bit05_StateFastStop := wMcMainStatusWord.5;
RxAndTxData.stMcMainStatusWord.Bit06_StateDisable := wMcMainStatusWord.6;
RxAndTxData.stMcMainStatusWord.Bit07_Warning := wMcMainStatusWord.7;
RxAndTxData.stMcMainStatusWord.Bit08_SpeedCtrlLimited := wMcMainStatusWord.8;
RxAndTxData.stMcMainStatusWord.Bit09_BusSelected := wMcMainStatusWord.9;
RxAndTxData.stMcMainStatusWord.Bit10_XnIsEqualToWn := wMcMainStatusWord.10;
RxAndTxData.stMcMainStatusWord.Bit11_WiqTLimited := wMcMainStatusWord.11;
RxAndTxData.stMcMainStatusWord.Bit12_XnIsEqualToZero := wMcMainStatusWord.12;
RxAndTxData.stMcMainStatusWord.Bit13_NCtrlenable := wMcMainStatusWord.13;
RxAndTxData.stMcMainStatusWord.Bit14_ExtrnalTorqueRelease := wMcMainStatusWord.14;
RxAndTxData.stMcMainStatusWord.Bit15_MainAliveToggle := wMcMainStatusWord.15;
///}}}

/// Copyng MC Auxiliary Status Word Into Structure {{{    
RxAndTxData.stMcAuxiliaryStatusWord.Bit00_FaultB := wMcAuxiliaryStatusWord.0;
RxAndTxData.stMcAuxiliaryStatusWord.Bit01_FaultC := wMcAuxiliaryStatusWord.1;
RxAndTxData.stMcAuxiliaryStatusWord.Bit02_FaultC := wMcAuxiliaryStatusWord.2;
RxAndTxData.stMcAuxiliaryStatusWord.Bit03_FaultDWarning := wMcAuxiliaryStatusWord.3;
RxAndTxData.stMcAuxiliaryStatusWord.Bit04_TrafoOvertempWarning := wMcAuxiliaryStatusWord.4;
RxAndTxData.stMcAuxiliaryStatusWord.Bit05_TrafoInsolationWarning := wMcAuxiliaryStatusWord.5;
RxAndTxData.stMcAuxiliaryStatusWord.Bit06_uu := wMcAuxiliaryStatusWord.6;
RxAndTxData.stMcAuxiliaryStatusWord.Bit07_uu := wMcAuxiliaryStatusWord.7;
RxAndTxData.stMcAuxiliaryStatusWord.Bit08_uu := wMcAuxiliaryStatusWord.8;
RxAndTxData.stMcAuxiliaryStatusWord.Bit09_uu := wMcAuxiliaryStatusWord.9;
RxAndTxData.stMcAuxiliaryStatusWord.Bit10_ThHSWarning := wMcAuxiliaryStatusWord.10;
RxAndTxData.stMcAuxiliaryStatusWord.Bit11_ThHSMaxWarning := wMcAuxiliaryStatusWord.11;
RxAndTxData.stMcAuxiliaryStatusWord.Bit12_ParSetBit00 := wMcAuxiliaryStatusWord.12;
RxAndTxData.stMcAuxiliaryStatusWord.Bit13_ParSetBit01 := wMcAuxiliaryStatusWord.13;
RxAndTxData.stMcAuxiliaryStatusWord.Bit14_ParSetBit02 := wMcAuxiliaryStatusWord.14;
RxAndTxData.stMcAuxiliaryStatusWord.Bit15_ParSetBit03 := wMcAuxiliaryStatusWord.15;        
///}}}

(*    
// Copyng Output Integer and real Structure Data into Global Variable
RxAndTxData.stLcMainStatusWord := stLcMainStatusWord;
RxAndTxData.stMcMainStatusWord := stMcMainStatusWord;
RxAndTxData.stLcAuxiliaryStatusWord := stLcAuxiliaryStatusWord;
RxAndTxData.stMcAuxiliaryStatusWord := stMcAuxiliaryStatusWord;
*)

END_FUNCTION_BLOCK

// ---- EventLogger/FunctionBlocks/FB_EventAlarm.TcPOU
FUNCTION_BLOCK FB_EventAlarm
VAR_INPUT
    bEvent         : BOOL;
    nEventID    : UDINT;
    sSource     : STRING;
END_VAR
VAR_OUTPUT
END_VAR
VAR
    bIsInitialized : BOOL;
    
    fbSourceInfo     : FB_TcSourceInfo;
    fbAlarm         : FB_TcAlarm;
    eventEntry        : TcEventEntry;
    fbRtEvent        : R_TRIG;
    fbFtEvent        : F_TRIG;
    
    hr                : HRESULT;
    hrLastError        : HRESULT;
END_VAR

(* Initialization *) 
    IF NOT bIsInitialized THEN
        bIsInitialized := TRUE;
        eventEntry := Tc_Events.MyEventClass.WarningEvent;
        eventEntry.nEventId := nEventID;
        
        fbSourceInfo.Clear();
        fbSourceInfo.sName := sSource;
        
        hr := fbAlarm.CreateEx(eventEntry, TRUE, ipSourceInfo := fbSourceInfo);
        
        IF FAILED(hr) THEN
            hrLastError := hr;
        END_IF
    END_IF
    
(* event trigger *)
    fbRtEvent(CLK := bEvent);
    fbFtEvent(CLK := bEvent);
    
(* alarm reised  *)
    IF fbRtEvent.Q THEN
        hr := fbAlarm.Raise(0);
        IF FAILED(hr) THEN
            hrLastError := hr;
        END_IF
    END_IF
    
(* alarm cleared *)
    IF fbFtEvent.Q THEN
        hr := fbAlarm.Clear(0, bResetConfirmation := TRUE);
        IF FAILED(hr) THEN 
            hrLastError := hr;
        END_IF
    END_IF

END_FUNCTION_BLOCK
